	// Populated ID identifies an item in the sorter
	// Between the two Divert status codes indicates that the item has attempted to divert
	IF ExitItemInSorter.ID <> '' THEN
		// Capture the Item encoder index and the Item at the current index
		//  This represents the first item record for this item
		//  It is captured to log the start index to allow this first record to be updated
		//  when the item is completely diverted
		IF ExitItemFound.Item.ID = '' THEN
			ExitItemFound.Counts := ExitSorterIndex;
			ExitItemFound.Item := ExitItemInSorter;
			IF ExitItemFound.Item.Status = E_StatusCode.Divert_Complete THEN
				ExitComplete := TRUE;
			END_IF
		END_IF
		// When ExitComplete is TRUE, and the ID's match, clear out this Item
		IF ExitComplete THEN
			IF ExitItemInSorter.ID = ExitItemFound.Item.ID THEN
				IF aItems[ExitSorterIndex].ID <> '' THEN
					IF .nSortBufferLogEnable.BUFFER_DUMP THEN
						sMessage := CONCAT(' Item: ', aItems[ExitSorterIndex].ID);
						sMessage := CONCAT(sMessage,' Index: ');
						sMessage := CONCAT(sMessage, UDINT_TO_STRING(ExitSorterIndex));
						sMessage := CONCAT(sMessage,' Item Status: ');
						sMessage := CONCAT(sMessage, DINT_TO_STRING(aItems[ExitSorterIndex].Status));
						sMessage := CONCAT(sMessage,' Item Ext Status: ');
						sMessage := CONCAT(sMessage, DINT_TO_STRING(aItems[ExitSorterIndex].ExtStatus));
						// Write to the Error List
						ADSLOGSTR( msgCtrlMask := ADSLOG_MSGTYPE_HINT OR ADSLOG_MSGTYPE_LOG
							, msgFmtStr := 'Exit Complete Dump Info: %s'
							, strArg := sMessage);
					END_IF
				END_IF
				aItems[ExitSorterIndex] := BlankItem;
			END_IF
		// When ExitComplete is FALSE, test for a diverting/diverted item
		ELSE
			// Detect when this item is in a diverting state
			IF (ExitItemInSorter.Status >= E_StatusCode.Diverting
			   OR ExitItemInSorter.Status <= E_StatusCode.Divert_Success)
			   THEN
			   	ExitInDivert := TRUE;
				(*
					Status value increase from Diverting to Divert_Complete
					Codes to indicate divert disposition are between Diverting and Divert_Detected
					Divert_Full and Diverting are set in FB_DivertDecision/FB_DivertControl
					Divert_Detected, Divert_Success, and Divert_Missed are set in FB_ConfirmCheck
				*)
				ExitDiverting := TRUE;
				IF ExitItemInSorter.Status = E_StatusCode.Divert_Detected THEN
					ExitDetected := TRUE;
				END_IF
				// Once the divert is successful, we are no longer "diverting"
				IF ExitItemInSorter.Status = E_StatusCode.Divert_Success THEN
					ExitSuccess := TRUE;
					ExitDiverting := FALSE;
				END_IF
				(*	
					ExitItemInSorter is the current item being examined
					ExitItemFound.Item is a copy of the Array item at ExitItemFound.Counts
					ExitItemFound.Counts references the Array index of the first record associated with this item
					When a Status/ExtStatus of greater value is detected, the first record Status/ExtStatus is overwritten
					The ExitItemFound.Item.Status/.ExtStatus is also updated
				*)
				IF ExitItemInSorter.Status > aItems[ExitItemFound.Counts].Status THEN
					aItems[ExitItemFound.Counts].Status := ExitItemInSorter.Status;
					ExitItemFound.Item.Status := ExitItemInSorter.Status;
				END_IF
				IF ExitItemInSorter.ExtStatus > aItems[ExitItemFound.Counts].ExtStatus THEN
					aItems[ExitItemFound.Counts].ExtStatus := ExitItemInSorter.ExtStatus;
					ExitItemFound.Item.ExtStatus := ExitItemInSorter.ExtStatus;
				END_IF
			END_IF
			aItems[ExitSorterIndex].Status := ExitItemFound.Item.Status;
		END_IF
	ELSE
		(*
			This path is followed when the ExitItemInSorter.ID is empty, which indicates
			that the array record associated with this index is not occupied

			ExitInDivert, ExitDiverting and ExitSuccess are all set while the .ID is not empty
		*)
		// This item was in a "diverting" state
		IF ExitInDivert THEN
			// This item is not currently diverting
			IF NOT ExitDiverting THEN
				// Only change to a Divert_Success if a Divert_Success was detected
				// Any other status is captured in the ELSE clause of the CASE statement
				IF ExitSuccess THEN
					ExitItemFound.Item.Status := E_StatusCode.Divert_Success;
				END_IF
				ExitItemFound.Item.CapturedInMetrics := TRUE;
				ExitItemFound.Item.MessageType := E_MessageIds.TransportComplete_26;
				fb_UpdateBuffer.AddItem(ExitItemFound.Item);
				aItems[ExitItemFound.Counts].Status := E_StatusCode.Divert_Complete;
			END_IF
		END_IF
		// Clear the last detected Exit item
		ExitItemFound.Item := BlankItem;
		// Reset the Detection booleans
		ExitInDivert := FALSE;
		ExitDiverting := FALSE;
		ExitDetected := FALSE;
		ExitSuccess := FALSE;
		ExitComplete := FALSE;
	END_IF
END_FOR

// If the ID is populated, we didn't find a match to update
IF st_ToUpdate.Item.ID <> '' THEN
	IF .nSortBufferLogEnable.BUFFER_UNASSIGNED THEN
		sMessage := CONCAT(' Item: ', st_ToUpdate.Item.ID);
		// Write to the Error List
		ADSLOGSTR( msgCtrlMask := ADSLOG_MSGTYPE_HINT OR ADSLOG_MSGTYPE_LOG
			, msgFmtStr := 'Item Not Updated: %s'
			, strArg := sMessage);
	END_IF
	st_ToUpdate.Item.Status := E_StatusCode.Assign_NotFound;
	st_ToUpdate.Item.DeviceID := st_Sorter.Config.Name;
	st_ToUpdate.Item.MessageType := E_MessageIds.TransportResponse_25;
	fb_UpDateBuffer.AddItem(st_ItemToAdd := st_ToUpdate.Item);
	st_ToUpdate.Item := BlankItem;
END_IF

END_PROGRAM

// ---- POUs/Sorter_P2150.TcPOU
PROGRAM Sorter_P2150

VAR_IN_OUT
	In_ItemToInduct					: ST_Item;
	In_InductingItem				: ST_Item;
	st_tempItem						: ST_ItemTemporary;	// Temporary record used when barcode not yet received
	{attribute 'OPC.UA.DA' := '0'}
	st_Sorter						: ST_Sorter;
	{attribute 'OPC.UA.DA' := '0'}
	aDiverts						: ARRAY[Sorter.DIVERTMIN_P2150..Sorter.NUMBEROFDIVERTS_P2150] OF ST_DIVERT;
	aItems 							: ARRAY[Sorter.SORTERENCODERMIN_P2150..Sorter.SORTERENCODERMAX_P2150] OF ST_Item;
END_VAR

VAR_INPUT
	DestinationOverride	: DINT;	// Pass in Divert to sent item to regardless of the direction received
	ItemsArrayMax		: UDINT;
	ItemsArrayMin		: UDINT;
	DivertArrayMax		: DINT;
	DivertArrayMin		: DINT;
END_VAR

VAR_OUTPUT
	st_DischargeItem	:	ST_Item;
END_VAR
VAR
	// Sorter Diagnostics
	aSorterDiagLog		: ST_ItemLogBuffer;
	fbSorterDiagLog		: FB_ItemLogBuffer;

	//Logging Variables
	UpdateSorterLog : FB_UpdateLog;
	
	//Induct Variables
	testEncoderCount		: UDINT;
	exitEncoderCount		: UDINT;
	lastCompareCount		: UDINT;
	updatingEncoderCount	: UDINT;

	tailendcount		: DINT := 0;
	inductindex 		: DINT;
	
	//Divert Variables
	{attribute 'OPC.UA.DA' := '0'}
	fb_DivertDecision 		: FB_DivertDecision;
	{attribute 'OPC.UA.DA' := '0'}
	fb_DivertFullMonitor  	: ARRAY[Sorter.DIVERTMIN_P2150..Sorter.NUMBEROFDIVERTS_P2150] OF FB_DivertFullMonitor;
	DivertIndex				: DINT;
	Divertoffset			: INT;
	nTestItemIndex			: UDINT;
	Output2ItemIndex		: UDINT;

	// Confirm Check variables
	fb_ConfirmCheck 		: ARRAY[Sorter.DIVERTMIN_P2150..Sorter.NUMBEROFDIVERTS_P2150] OF FB_ConfirmCheck;
	st_ConfirmItem 			: ARRAY[Sorter.DIVERTMIN_P2150..Sorter.NUMBEROFDIVERTS_P2150] OF ST_Item;
	nConfirmItemIndex 		: UDINT;
	
	workingItem			: ST_Item;	// Actual item to induct

	LastItemInducted 	: STRING;
	nIndexToClear		: UDINT;	// Clear Item Array at this index
	nItemArraySize		: UDINT;

	rInductPE			: R_TRIG; 	// Capture the Rising edge of the Induct PE
	fInductPE			: F_TRIG; 	// Capture the Falling edge of the Induct PE
	sMessage			: STRING;

	st_DisplayItem		:st_Item;
	
	LogSorterDump: BOOL := FALSE;

	fb_FindDestination		: FB_FindDestination;
	{attribute 'OPC.UA.DA' := '0'}
	aTempDiverts			: ARRAY[Sorter.DIVERTMIN_P2150..Sorter.NUMBEROFDIVERTS_P2150] OF ST_DIVERT;

	nItemBufferLogEnable	:	UDINT;
	nSorterLogEnable		:	UDINT;
	nDivertLogEnable		:	UDINT;
	nSortBufferLogEnable	:	UDINT;
END_VAR

nItemBufferLogEnable := GVL_Logging.nItemBufferLogEnable OR GVL_Logging.nItemBufferLogEnableP2150;
nSorterLogEnable := GVL_Logging.nSorterLogEnable OR GVL_Logging.nSorterLogEnableP2150;
nDivertLogEnable := GVL_Logging.nDivertLogEnable OR GVL_Logging.nDivertLogEnableP2150;
nSortBufferLogEnable := GVL_Logging.nSortBufferLogEnable OR GVL_Logging.nSortBufferLogEnableP2150;
aTempDiverts := aDiverts;

// Initialize FB_ItemExtBuffer
fbSorterDiagLog(st_BufferData := aSorterDiagLog);

(*
// Test visu variables	
inductPE := SorterInductPE;
ItemsOut := Items;
ArrivalOut := ArrivalBuffer;
// End test variables
*)
(*
	Capture the Upper/Lower bound of relevant IO_OUT arrays for looping purposes
	ItemsArrayMax/Min for the sorter array slot count
*)
// Size is Max - Min + 1 to capture both extremes
nItemArraySize := ItemsArrayMax - ItemsArrayMin + 1;

FOR divertIndex := DivertArrayMin TO DivertArrayMax DO
	fb_DivertFullMonitor[DivertIndex](Divert := aDiverts[divertIndex]);
END_FOR

(*
	Detect barcode receipt after item is already in Item array
	the tempItem is reset when the induct PE is cleared
	The tempItem is populated when the induct PE is blocked and there
	is not an associated barcode waiting to be inducted
*)
IF st_tempItem.Item.ID <> '' THEN
	// Test the IN_ItemToInduct.ID for a value
	// This record will be cleared as soon as it reaches the sorter loop
	IF In_ItemToInduct.ID <> '' THEN
		// The tempItem is overwritten with the IN_ItemToInduct after it is updated
		// But the starting encoder count is not changed so the same items can be updated
		// if the destination update is received while the item is still being inducted
		IF In_ItemToInduct.ID <> st_tempItem.Item.ID THEN 
			// Set the starting count for the testing/updating process
			// The testEncodeCount is incremented upon start, so we start -1 of the encoder count for the item
			testEncoderCount := f_CalculateIndex(Offset := -1, InitialValue:= st_tempItem.Counts, BufferSize := nItemArraySize);
			// Clear the length and start over
			In_ItemToInduct.Length := 0;
			st_tempItem.Item := In_ItemToInduct;
		END_IF 
		// Test for a change of destination after the barcode data has been received
		IF In_ItemToInduct.Destination <> st_tempItem.Item.Destination THEN 
			// Set the starting count for the testing/updating process
			// The testEncodeCount is incremented upon start, so we start -1 of the encoder count for the item
			testEncoderCount := f_CalculateIndex(Offset := -1, InitialValue:= st_tempItem.Counts, BufferSize := nItemArraySize);
			// Clear the length and start over
			In_ItemToInduct.Length := 0;
			// Copy the IN_ItemToInduct to prevent running this until something else in the record changes
			st_tempItem.Item := IN_ItemToInduct;
		END_IF
	END_IF 
END_IF


// Test for the rising edge of the induct PE
// Use this rising edge to log the IN_ItemToInduct record
rInductPE(CLK:= st_Sorter.InductPE, Q =>);

IF rInductPE.Q THEN
	IF nSorterLogEnable.SORTER_INDUCT THEN
		sMessage := CONCAT('Item: ', In_ItemToInduct.ID);
		sMessage := CONCAT(sMessage, ' Pulses: ');
		sMessage := CONCAT(sMessage, UDINT_TO_STRING(st_Sorter.EncoderCounts));
		// Write to the Error List
		ADSLOGSTR( msgCtrlMask := ADSLOG_MSGTYPE_HINT OR ADSLOG_MSGTYPE_LOG
			, msgFmtStr := CONCAT(st_sorter.Config.Name, ' Induct Info: %s')
			, strArg := sMessage);
	END_IF
END_IF
// Test for the falling edge of the induct PE
// Use this falling edge to clear the IN_ItemToInduct record
fInductPE(CLK:= st_Sorter.InductPE, Q =>);

IF fInductPE.Q THEN
	IF nSorterLogEnable.SORTER_INDUCT THEN
		sMessage := CONCAT('Item: ', In_ItemToInduct.ID);
		sMessage := CONCAT(sMessage,' Pulses: ');
		sMessage := CONCAT(sMEssage, UDINT_TO_STRING(st_Sorter.EncoderCounts));
		// Write to the Error List
		ADSLOGSTR( msgCtrlMask := ADSLOG_MSGTYPE_HINT OR ADSLOG_MSGTYPE_LOG
			, msgFmtStr := CONCAT(st_sorter.Config.Name, ' Cleared Induct Info: %s')
			, strArg := sMessage);
	END_IF
	// Clear the record
	In_InductingItem :=  BlankItem;
END_IF

// Process every array index between the current index and the last processed index
WHILE st_Sorter.EncoderCounts <> testEncoderCount DO

	// Capture the lastEncoderCount before changing it for comparison of last inducted items
	lastCompareCount := testEncoderCount;

	// Increment the testEncoderCount
	// The testEncoderCount variable will be used throughout the processing to ensure
	//	that all array elements are processed
	testEncoderCount := f_CalculateIndex(Offset := 1, InitialValue:= testEncoderCount, BufferSize := nItemArraySize);
	IF st_Sorter.InductPE THEN
	  	IF (In_ItemToInduct.ID <> '') THEN
			In_InductingItem := In_ItemToInduct;
			In_ItemToInduct := BlankItem;
			// If there is an override, use the value as the destination
			IF DestinationOverride <> 0 THEN
				IF nSorterLogEnable.SORTER_DESTINATION_LU THEN
					sMessage := CONCAT(' Orig: ', DINT_TO_STRING(In_InductingItem.Destination));
					sMessage := CONCAT(sMessage, 'New: ');
					sMessage := CONCAT(sMessage, DINT_TO_STRING(DestinationOverride));
					// Write to the Error List
					ADSLOGSTR( msgCtrlMask := ADSLOG_MSGTYPE_HINT OR ADSLOG_MSGTYPE_LOG
						, msgFmtStr := CONCAT(st_sorter.Config.Name, ' DestinationOverride %s')
						, strArg := sMessage);
				END_IF
				In_InductingItem.Destination := DestinationOverride;
			END_IF
			IF nSorterLogEnable.SORTER_DESTINATION_LU THEN
				sMessage := CONCAT('Destination: ', DINT_TO_STRING(In_InductingItem.Destination));
				// Write to the Error List
				ADSLOGSTR( msgCtrlMask := ADSLOG_MSGTYPE_HINT OR ADSLOG_MSGTYPE_LOG
					, msgFmtStr := CONCAT(st_sorter.Config.Name, ' Sorter Lookup %s')
					, strArg := sMessage);
			END_IF
			fb_FindDestination(RoundRobin := st_Sorter.RoundRobin
							, SorterLogEnable := nSorterLogEnable
							, aDiverts := aTempDiverts
							, DestinationID := In_InductingItem.Destination
							, DestinationIndex => In_InductingItem.DestinationIdx);
			IF nSorterLogEnable.SORTER_INDUCT_PE THEN
				sMessage := CONCAT('Item: ', In_InductingItem.ID);
				sMessage := CONCAT(sMessage,' Pulses: ');
				sMessage := CONCAT(sMessage, UDINT_TO_STRING(st_Sorter.EncoderCounts));
				sMessage := CONCAT(sMessage,' Dest: ');
				sMessage := CONCAT(sMessage, DINT_TO_STRING(In_InductingItem.Destination));
				sMessage := CONCAT(sMessage,' DestIdx: ');
				sMessage := CONCAT(sMessage, DINT_TO_STRING(In_InductingItem.DestinationIdx));
				// Write to the Error List
				ADSLOGSTR( msgCtrlMask := ADSLOG_MSGTYPE_HINT OR ADSLOG_MSGTYPE_LOG
					, msgFmtStr := CONCAT(st_sorter.Config.Name, ' Inducting Info: %s')
					, strArg := sMessage);
			END_IF
		END_IF
	  	IF (In_InductingItem.ID <> '') THEN
			LastItemInducted := In_InductingItem.ID;
			IF aItems[testEncoderCount].ID <> '' THEN
				IF aItems[testEncoderCount].Status >= E_StatusCode.Diverting AND aItems[testEncoderCount].Status <= E_StatusCode.Divert_UnknownError THEN
					aItems[testEncoderCount].Status := E_StatusCode.Divert_UnknownError;
				END_IF
				UpdateSorterLog(Status := aItems[testEncoderCount].Status, ItemID := aItems[testEncoderCount].UniqueID);
			END_IF
		
			// Set the Item status
			In_InductingItem.Status := E_StatusCode.In_Sorter;

			// Check for destination full on the first pass, then ignore it.
			IF In_InductingItem.Length = 0 AND DestinationOverride = 0 THEN
				IF aDiverts[In_InductingItem.DestinationIdx].Full AND DestinationOverride = 0 THEN
					IF st_Sorter.Config.RecircUsed THEN
						In_InductingItem.Destination := st_Sorter.Config.RecircDestination;
						In_InductingItem.DestinationIdx := st_Sorter.Config.RecircDestIdx;
						In_InductingItem.ExtStatus := E_StatusCode.Divert_Recirculated;
					ELSE
						In_InductingItem.Destination := st_Sorter.Config.DefaultDestination;
						In_InductingItem.DestinationIdx := st_Sorter.Config.DefaultDestIdx;
						In_InductingItem.ExtStatus := E_StatusCode.Divert_Full;
					END_IF
				END_IF
			END_IF
			// Clear the extend counter
			tailendcount := 0;

			// Copy the ItemToInduct to the WorkingItem that will be inducted
			workingItem := In_InductingItem;
			// Increment the Length on the ItemToInduct record, then it will be added to the array
			//  and the length will increment
			In_InductingItem.Length := In_InductingItem.Length +  1;
			// Determined by UniqueID = 0
		ELSE //If the item makes it to the sorter, but is not identified, induct the item with tempItem.Item
			LastItemInducted := 'UNKNOWN';
			UpdateSorterLog(Status := E_StatusCode.UnidentifiedItem, ItemID := st_tempItem.Item.UniqueID);

			// Process this the first time
			IF st_tempItem.Item.Length = 0 THEN
				IF nSorterLogEnable.SORTER_INDUCT_PE THEN
					sMessage := CONCAT('Temp Item: ', st_tempItem.Item.ID);
					sMessage := CONCAT(sMessage,' Pulses: ');
					sMessage := CONCAT(sMessage, UDINT_TO_STRING(st_Sorter.EncoderCounts));
					sMessage := CONCAT(sMessage,' Dest: ');
					sMessage := CONCAT(sMessage, DINT_TO_STRING(st_tempItem.Item.Destination));
					sMessage := CONCAT(sMessage,' DestIdx: ');
					sMessage := CONCAT(sMessage, DINT_TO_STRING(st_tempItem.Item.DestinationIdx));
					sMessage := CONCAT(sMessage,' Length: ');
					sMessage := CONCAT(sMessage, DINT_TO_STRING(st_tempItem.Item.Length));
					// Write to the Error List
					ADSLOGSTR( msgCtrlMask := ADSLOG_MSGTYPE_HINT OR ADSLOG_MSGTYPE_LOG
						, msgFmtStr := CONCAT(st_sorter.Config.Name, ' Inducting Info: %s')
						, strArg := sMessage);
				END_IF
				IF aDiverts[st_Sorter.Config.DefaultDestIdx].Full THEN
					IF st_Sorter.Config.RecircUsed THEN
						st_tempItem.Item.Destination := st_Sorter.Config.RecircDestination;
						st_tempItem.Item.DestinationIdx := st_Sorter.Config.RecircDestIdx;
						st_tempItem.Item.ExtStatus := E_StatusCode.Divert_Recirculated;
					ELSE
						st_tempItem.Item.Destination := st_Sorter.Config.DefaultDestination;
						st_tempItem.Item.DestinationIdx := st_Sorter.Config.DefaultDestIdx;
						st_tempItem.Item.ExtStatus := E_StatusCode.Divert_Full;
					END_IF
				ELSE
					IF DestinationOverride = 0 THEN
						st_tempItem.Item.Destination := st_Sorter.Config.DefaultDestination;
					ELSE
						st_tempItem.Item.Destination := DestinationOverride;
					END_IF
					IF nSorterLogEnable.SORTER_DESTINATION_LU THEN
						sMessage := CONCAT('Destination: ', DINT_TO_STRING(st_tempItem.Item.Destination));
						// Write to the Error List
						ADSLOGSTR( msgCtrlMask := ADSLOG_MSGTYPE_HINT OR ADSLOG_MSGTYPE_LOG
							, msgFmtStr := CONCAT(st_sorter.Config.Name, ' Temp Lookup %s')
							, strArg := sMessage);
					END_IF
					fb_FindDestination(RoundRobin := st_Sorter.RoundRobin
							, SorterLogEnable := nSorterLogEnable
							, aDiverts := aTempDiverts
							, DestinationID := st_tempItem.Item.Destination
							, DestinationIndex => st_tempItem.Item.DestinationIdx);
				END_IF		
				IF nSorterLogEnable.SORTER_INDUCT_PE THEN
					sMessage := CONCAT('Temp Item: ', st_tempItem.Item.ID);
					sMessage := CONCAT(sMessage,' Pulses: ');
					sMessage := CONCAT(sMessage, UDINT_TO_STRING(st_Sorter.EncoderCounts));
					sMessage := CONCAT(sMessage,' Dest: ');
					sMessage := CONCAT(sMessage, DINT_TO_STRING(st_tempItem.Item.Destination));
					sMessage := CONCAT(sMessage,' DestIdx: ');
					sMessage := CONCAT(sMessage, DINT_TO_STRING(st_tempItem.Item.DestinationIdx));
					// Write to the Error List
					ADSLOGSTR( msgCtrlMask := ADSLOG_MSGTYPE_HINT OR ADSLOG_MSGTYPE_LOG
						, msgFmtStr := CONCAT(st_sorter.Config.Name, ' Inducting Info: %s')
						, strArg := sMessage);
				END_IF
			END_IF
			// Copy the tempItem.Item to the WorkingItem that will be inducted
			workingItem := st_tempItem.Item;
			// Increment the Length on the ItemToInduct record, then it will be added to the array
			//  and the length will increment
			st_tempItem.Item.Length := st_tempItem.Item.Length +  1;
		END_IF

		// Induct everything
		aItems[testEncoderCount] := workingItem;
		fbSorterDiagLog.AddItem(workingItem);
	// Follow this path when the induct photo-eye is cleared
	ELSE
		// Extend the end of the item by a set amount, or to a mimimum length
		// Test to verify that the Item index is clear, and we are still extending the length of the item
		IF aItems[lastCompareCount].ID <> '' THEN
			IF tailendcount < st_Sorter.Config.TailEndLength AND st_Sorter.Config.TailEndLength > 0 THEN
				aItems[testEncoderCount] := aItems[lastCompareCount]; 
				fbSorterDiagLog.AddItem(aItems[lastCompareCount]);
				aItems[testEncoderCount].Length := aItems[testEncoderCount].Length + 1;
				tailendcount := tailendcount + 1;
			END_IF
			IF aItems[lastCompareCount].Length < st_Sorter.Config.MinimumLength AND st_Sorter.Config.MinimumLength > 0 THEN
				aItems[testEncoderCount] := aItems[lastCompareCount]; 
				fbSorterDiagLog.AddItem(aItems[lastCompareCount]);
				aItems[testEncoderCount].Length := aItems[testEncoderCount].Length + 1;
			END_IF
		END_IF
	END_IF
END_WHILE

// Process every array index between the current index and the last processed exit index
WHILE st_Sorter.EncoderCounts <> exitEncoderCount DO

	// Increment the exitEncoderCount
	// The exitEncoderCount variable will be used throughout the processing to ensure
	//	that all array elements are processed
	exitEncoderCount := f_CalculateIndex(Offset := 1, InitialValue:= exitEncoderCount, BufferSize := nItemArraySize);
	// Process the diverts relative to the current encoder count
	FOR divertIndex := DivertArrayMin TO DivertArrayMax DO
		// Get the distance to each divert, distance is the number of pulses to actuation
		Divertoffset := aDiverts[divertIndex].Config.Distance;
		// Calculate the index of the item to test for a divert
		// Subtract the offset from the current encoder count (exitEncoderCount)
		// As the encoder count increases, the current index pointer advances
		// Subtracting looks backwards into the sorter item array to test for items at the diverts
		//	distance that should be diverted
		nTestItemIndex := F_CalculateIndex(initialvalue := exitEncoderCount
										, offset := -(Divertoffset)
										, BufferSize := (ItemsArrayMax + 1));	
		//Setup Out2Item for energizing 2nd divert output
		Output2ItemIndex := F_CalculateIndex(initialvalue := exitEncoderCount
										, offset := -(Divertoffset + UINT_TO_INT(st_Sorter.Config.Output2Offset))
										, BufferSize := (ItemsArrayMax + 1));	
		// Log Diverts
		IF aItems[nTestItemIndex].DestinationIdx = divertIndex THEN
			IF nSorterLogEnable.SORTER_DIVERTS THEN
				sMessage := CONCAT('Item: ', aItems[nTestItemIndex].ID);
				sMessage := CONCAT(sMessage,' Index: ');
				sMessage := CONCAT(sMessage, UDINT_TO_STRING(nTestItemIndex));
				sMessage := CONCAT(sMessage,' Dest: ');
				sMessage := CONCAT(sMessage, DINT_TO_STRING(aItems[nTestItemIndex].Destination));
				sMessage := CONCAT(sMessage,' DestIdx: ');
				sMessage := CONCAT(sMessage, DINT_TO_STRING(aItems[nTestItemIndex].DestinationIdx));
				sMessage := CONCAT(sMessage,' Divert Status: ');
				sMessage := CONCAT(sMessage, DINT_TO_STRING(aDiverts[DivertIndex].Status));
				sMessage := CONCAT(sMessage,' Item Status: ');
				sMessage := CONCAT(sMessage, DINT_TO_STRING(aItems[nTestItemIndex].Status));
				// Write to the Error List
				ADSLOGSTR( msgCtrlMask := ADSLOG_MSGTYPE_HINT OR ADSLOG_MSGTYPE_LOG
					, msgFmtStr := CONCAT(st_sorter.Config.Name, ' Item at Divert Index: %s')
					, strArg := sMessage);
			END_IF
		END_IF
		fb_DivertDecision( bLog := nDivertLogEnable.DIVERT_DECISION 
					 , Output1Item		:= aItems[nTestItemIndex]
					 , Output2Item		:= aItems[Output2ItemIndex]
					 , Divert 			:= aDiverts[DivertIndex]
					 , DivertIndex		:= DivertIndex
					 );
		// Calculate the distance to the confirm PE to test for a successful divert
		nConfirmItemIndex := F_CalculateIndex(initialvalue := exitEncoderCount
										, offset := -(Divertoffset + aDiverts[divertIndex].Config.ConfirmDist)
										, BufferSize := (ItemsArrayMax + 1));
		// Log Confirms
		IF aItems[nConfirmItemIndex].Status >= E_StatusCode.Diverting
		   AND aItems[nConfirmItemIndex].Status <= E_StatusCode.Divert_Complete
		   AND aItems[nConfirmItemIndex].UniqueID <> 0
		   AND aItems[nConfirmItemIndex].DestinationIdx = DivertIndex
		   THEN
			IF nSorterLogEnable.SORTER_CONFIRMS THEN
				sMessage := CONCAT('Item: ', aItems[nConfirmItemIndex].ID);
				sMessage := CONCAT(sMessage,' Index: ');
				sMessage := CONCAT(sMessage, UDINT_TO_STRING(nConfirmItemIndex));
				sMessage := CONCAT(sMessage,' Dest: ');
				sMessage := CONCAT(sMessage, DINT_TO_STRING(aItems[nConfirmItemIndex].Destination));
				sMessage := CONCAT(sMessage,' DestIdx: ');
				sMessage := CONCAT(sMessage, DINT_TO_STRING(aItems[nConfirmItemIndex].DestinationIdx));
				sMessage := CONCAT(sMessage,' Divert Status: ');
				sMessage := CONCAT(sMessage, DINT_TO_STRING(aDiverts[DivertIndex].Status));
				sMessage := CONCAT(sMessage,' Item Status: ');
				sMessage := CONCAT(sMessage, DINT_TO_STRING(aItems[nTestItemIndex].Status));
				// Write to the Error List
				ADSLOGSTR( msgCtrlMask := ADSLOG_MSGTYPE_HINT OR ADSLOG_MSGTYPE_LOG
					, msgFmtStr := CONCAT(st_sorter.Config.Name, ' Item at Confirm Index: %s')
					, strArg := sMessage);
			END_IF
		END_IF
		fb_ConfirmCheck[divertIndex] ( bLog := nDivertLogEnable.DIVERT_DECISION 
					 , ConfirmItem		:= aItems[nConfirmItemIndex]
					 , ConfirmPE 		:= aDiverts[DivertIndex].ConfirmPE
					 , DivertIndex		:= DivertIndex
					 , bIsDischarge		:= aDiverts[DivertIndex].Config.IsDischarge
					 , DetectedItem => st_ConfirmItem[DivertIndex]
					 );
	END_FOR
	
	// Capture the last item discharged by this sorter section
	IF st_ConfirmItem[DivertArrayMax].ID <> '' THEN
		st_DischargeItem := st_ConfirmItem[DivertArrayMax];
	END_IF

	// Clear the Item array ahead of the current encoder count
	nIndexToClear := f_CalculateIndex(Offset := 40, InitialValue:= exitEncoderCount, BufferSize := nItemArraySize);
	IF aItems[nIndexToClear].ID <> '' THEN
		IF nSorterLogEnable.SORTER_DUMP THEN
			sMessage := CONCAT('Item: ', aItems[nIndexToClear].ID);
			sMessage := CONCAT(sMessage,' Index: ');
			sMessage := CONCAT(sMessage, UDINT_TO_STRING(nIndexToClear));
			sMessage := CONCAT(sMessage,' Item Status: ');
			sMessage := CONCAT(sMessage, DINT_TO_STRING(aItems[nIndexToClear].Status));
			sMessage := CONCAT(sMessage,' Destination: ');
			sMessage := CONCAT(sMessage, DINT_TO_STRING(aItems[nIndexToClear].Destination));
			sMessage := CONCAT(sMessage,' DestIndex: ');
			sMessage := CONCAT(sMessage, DINT_TO_STRING(aItems[nIndexToClear].DestinationIDX));
			// Write to the Error List
			ADSLOGSTR( msgCtrlMask := ADSLOG_MSGTYPE_HINT OR ADSLOG_MSGTYPE_LOG
				, msgFmtStr := CONCAT(st_sorter.Config.Name, ' Clear Ahead Dump Info: %s')
				, strArg := sMessage);
		END_IF
	END_IF
	aItems[nIndexToClear] := BlankItem;

END_WHILE

END_PROGRAM

// ---- POUs/MsgControl.TcPOU
PROGRAM MsgControl
VAR_INPUT
	TransmitEnable 				: BOOL;
	nConnectionIndex			: UDINT	:= 1;
END_VAR
VAR
	MsgID						: DINT;			// TCP/IP Message ID as per Communication protocol defined in FA 
	DeviceID					: STRING(5);	// TCP/IP Device ID as per Communication protocol defined in FA 
	BarCode						: STRING(20);	// TCP/IP Load ID (Bar Code) as per Communication protocol defined in FA
	BarCodeNoSpace				: STRING(20);	// TCP/IP Load ID (Bar Code) as per Communication protocol defined in FA stripped of spaces  
	Destination					: DINT;			// TCP/IP Destination as per Communication protocol defined in FA
	DefDestination				: DINT;			// TCP/IP Default Destination as per Communication protocol defined in FA
	Status						: BYTE;				// 
	Msg_EquipStatArry			: ARRAY[1..7] OF ST_Msg_EquipStat;
	nSystemStatusIndex 			: DINT; 	// Index used for Processing the system status array
	nTempOperState 				: DINT;	//Capture the Temporary Operating State of the Equipment for comparison
	nEquipStatusIndex			: DINT;	//Index used for adding items to the MSG_EquipStatArray
	StrStartPos					: INT;
	StrEndPos					: INT;
	MsgString					: STRING(55);
	RawMsgArray					: ARRAY[1..10] OF T_MaxString;	// Capture the last Raw messages for troubleshooting
	RawMsgLenArray				: ARRAY[1..10] OF INT;			// Capture the last  Raw message lengths for troubleshooting
	RawMsgStartPosArray			: ARRAY[1..10] OF INT;			// Capture the last  Raw message start positions for troubleshooting
	RawMsgEndPosArray			: ARRAY[1..10] OF INT;			// Capture the last  Raw message end positions for troubleshooting
	MsgArray					: ARRAY[1..10] OF STRING(55);		// Capture the last 10 messages that have been stripped from the starting character  for troubleshooting
	Blank_Msg_ConveyorStatArry	: ARRAY [1..7] OF ST_Msg_EquipStat := [7((Status := 99))];

	i 							: INT;
	j							: INT;
	
	RxCounter_Old				: UDINT;
	TxCounter_Old				: UDINT;
	TransmitMsgBuffer			: ARRAY [1..TransmitMsgBuffer_Size] OF STRING(55);	// Buffer to hold transmit messages
	TransmitMsgBuffer_Index		: INT :=	1;		// Index to the Buffer
	TransmitMsgStatus			: INT;			
	SendingMsg_Index			: INT :=	1;		// Index to send message
	
	ItemTransport				: ST_Item;		// Output Item Update with destination from ARUP Host (Send to Sorter PLC)
	BlankItem					: ST_Item := (ID := '', UniqueID := 0
													, Destination := 0
													, Status := E_StatusCode.No_Status
													, ExtStatus := E_StatusCode.No_Status
													, DeviceID := ''
													, MessageType := E_MessageIds.NoMessage_00);

	ReadBCRID_S2140_01_Old			: UDINT;		// Bar Code watch variable
	ReadBCRID_S2141_01_Old			: UDINT;		// Bar Code watch variable
	ReadBCRID_S2150_01_Old			: UDINT;		// Bar Code watch variable	
	ReadBCRID_S3080_01_Old			: UDINT;		// Bar Code watch variable
			
	TransmittedArray			: ARRAY[0..10] OF STRING(55);
	x							: DINT;
	y							: INT;
	
	SpacePosition				: INT;
	
	fb_CheckStopRegister		: FB_ManageCodes;	// Used to test for a specific Stop Code to report to the Host
	bOverHeight					: BOOL; 	// Detect OverHeight to report to the Host
	st_UpdateMessageToSend		: ST_Item;			// Message to Send to Host

	fb_SorterUpdateBuffer			: FB_ItemBuffer;	// Function to Process the SorterUpdateBuffer

	fb_SorterTransportBuffer_P2140	: FB_ItemBuffer;	// Function to Process the SorterTransportBuffer
	fb_SorterTransportBuffer_P2150	: FB_ItemBuffer;	// Function to Process the SorterTransportBuffer

	sMessage	:	STRING;
	
END_VAR

VAR CONSTANT
	SEND_ARRIVAL			:	INT := 5;
	SEND_LOCATION			:	INT := 7;
	TransmitMsgBuffer_Size	:	INT :=	25;		// Number of Messages to hold in buffer
END_VAR

// Create instances of Buffer Processing Functions to initialize the buffers and data
fb_SorterUpdateBuffer.Master := TRUE;
fb_SorterTransportBuffer_P2140.Master := TRUE;
fb_SorterTransportBuffer_P2150.Master := TRUE;

// Activate or de-activate logging
fb_SorterUpdateBuffer.LogEntries := .nItemBufferLogEnable.UPDATE OR .nItemBufferLogEnableP2150.UPDATE OR .nItemBufferLogEnableP2150.UPDATE;
fb_SorterTransportBuffer_P2140.LogEntries := .nItemBufferLogEnable.TRANSPORT OR .nItemBufferLogEnableP2140.TRANSPORT;
fb_SorterTransportBuffer_P2150.LogEntries := .nItemBufferLogEnable.TRANSPORT OR .nItemBufferLogEnableP2150.TRANSPORT;

// Setup Buffer names for Logging purposes
fb_SorterUpdateBuffer.Name := 'SYS UPDATE';
fb_SorterTransportBuffer_P2140.Name := 'P2140 SYS TRANSPORT';
fb_SorterTransportBuffer_P2150.Name := 'P2150 SYS TRANSPORT';

fb_SorterUpdateBuffer(st_BufferData := st_SorterUpdateBuffer
					, st_BufferFdbkIn := st_UpdateFdbkIn
					, st_BufferFdbkOut => st_UpdateFdbkOut);
fb_SorterTransportBuffer_P2140(st_BufferData := st_SorterTransportBuffer_P2140
					, st_BufferFdbkIn := st_TransportFdbkIn_P2140
					, st_BufferFdbkOut => st_TransportFdbkOut_P2140);
fb_SorterTransportBuffer_P2150(st_BufferData := st_SorterTransportBuffer_P2150
					, st_BufferFdbkIn := st_TransportFdbkIn_P2150
					, st_BufferFdbkOut => st_TransportFdbkOut_P2150);

(* -------------------- On Receive Message Process the data -------------------- *)
IF RxCounter_Old <> ServerControl.fbServer.aApplications[nConnectionIndex].RxCounter  THEN
	ItemTransport := BlankItem; // Clear the ItemTransport each pass to capture only new transport commands
	RECEIVE();
	// Test the DeviceID and route the Transport accordingly
	//	If there is only one possible DeviceID, this IF statement can be removed, but the fb_(TransportBuffer).AddItem call still has to be made
	//	Also, the default destination needs to be passed per DeviceID
	IF DeviceID = Sorter.st_Sorter_P2140Cfg.EquipID THEN
		fb_SorterTransportBuffer_P2140.AddItem(st_ItemToAdd := ItemTransport);
		P2140_DefaultDestination := DefDestination;
	END_IF
	IF DeviceID = Sorter.st_Sorter_P2150Cfg.EquipID THEN
		fb_SorterTransportBuffer_P2150.AddItem(st_ItemToAdd := ItemTransport);
		P2150_DefaultDestination := DefDestination;
	END_IF

	RxCounter_Old := ServerControl.fbServer.aApplications[nConnectionIndex].RxCounter;
END_IF

(* -------------------- Transmit Messages if any are waiting in the buffer --------------------- *)
IF SendingMsg_Index <> TransmitMsgBuffer_Index THEN
	TRANSMIT(TransmitEnable:= TRUE);
END_IF

(* -------------------- Watch Bar code readers and send message when load is read -------------------- *)
(* ----- BCR_S2140_01: P2140 Divert  ----- *)	
ReadBCRID_S2140_01_Old := BarCodeMessage(cDatamanReader := BarCodeReaders.BCR_S2140_01
									, nOldCount := ReadBCRID_S2140_01_Old
									, nMessageToSend := SEND_ARRIVAL);
(* ----- BCR_S2141_01: P2143 Induct Confirm ----- *)	
ReadBCRID_S2141_01_Old := BarCodeMessage(cDatamanReader := BarCodeReaders.BCR_S2141_01
									, nOldCount := ReadBCRID_S2141_01_Old
									, nMessageToSend := SEND_LOCATION);
(* ----- BCR_S2150_01: P2150 Sorter ----- *)	
ReadBCRID_S2150_01_Old := BarCodeMessage(cDatamanReader := BarCodeReaders.BCR_S2150_01
									, nOldCount := ReadBCRID_S2150_01_Old
									, nMessageToSend := SEND_ARRIVAL);
(* ----- BCR_S3080_01: P3080 Lane Confirm ----- *)	
ReadBCRID_S3080_01_Old := BarCodeMessage(cDatamanReader := BarCodeReaders.BCR_S3080_01
									, nOldCount := ReadBCRID_S3080_01_Old
									, nMessageToSend := SEND_LOCATION);


(* -------------------- Watch Sorter and Device Status and transmit on change -------------------- *)
// Transmit On update from Sorter
// Detect a new message to process when the in and out pointer values disagree
IF st_SorterUpdateBuffer.nInPointer <> fb_SorterUpdateBuffer.OutPointer THEN
	// Pull the next message out of the buffer
	fb_SorterUpdateBuffer.RemoveItem(st_ItemToReturn => st_UpdateMessageToSend);
	CASE st_UpdateMessageToSend.MessageType OF

		E_MessageIds.TransportResponse_25:			// Response to a Transport Command

			CASE st_UpdateMessageToSend.Status OF
				E_StatusCode.Assign_Accepted:		// Assignment Accepted
					TransmitMsgStatus := E_TransportResponse.Accepted; 
				E_StatusCode.Assign_Full:			// Assigned Lane Unavailable
					TransmitMsgStatus := E_TransportResponse.DivertLaneUnavailable; 
				E_StatusCode.Assign_NotFound:		// Assigned Load ID Not Found
					TransmitMsgStatus := E_TransportResponse.LoadIdNotFound; 
				E_StatusCode.Assign_NotInducted:	// Assigned Load Not Inducted
					TransmitMsgStatus := E_TransportResponse.NextLoadReady; 
				E_StatusCode.Diverting:	// Assigned Load already Inducting
					TransmitMsgStatus := E_TransportResponse.LateInduction; 
			ELSE
				TransmitMsgStatus := E_TransportResponse.UnknownFailure; // Capture any other failures
				IF nMessageLogEnable.TransportResponse_25 THEN
					sMessage := CONCAT(' Item: ', st_UpdateMessageToSend.ID);
					sMessage := CONCAT(sMessage,' Destination: ');
					sMessage := CONCAT(sMessage, DINT_TO_STRING(st_UpdateMessageToSend.Destination));
					sMessage := CONCAT(sMessage,' TR Status: ');
					sMessage := CONCAT(sMessage, DINT_TO_STRING(st_UpdateMessageToSend.Status));
					// Write to the Error List
					ADSLOGSTR( msgCtrlMask := ADSLOG_MSGTYPE_HINT OR ADSLOG_MSGTYPE_LOG
						, msgFmtStr := 'Unhandled Transport Response Status: %s'
						, strArg := sMessage);
				END_IF
			END_CASE
			TransmitMsgBuffer[TransmitMsgBuffer_Index] := TransportResponse(Device := st_UpdateMessageToSend.DeviceID
																			, Barcode := st_UpdateMessageToSend.ID
																			, Status := TransmitMsgStatus);
			TransmitMsgBuffer_Index := IncIndex(TransmitMsgBuffer_Index,1,TransmitMsgBuffer_Size);

		E_MessageIds.TransportComplete_26:			// Indication of the final disposition of a transported item

			CASE st_UpdateMessageToSend.Status OF
				E_StatusCode.Divert_Success:		// Divert Success Message
					TransmitMsgStatus := E_TransportComplete.Success; 
				E_StatusCode.Divert_Complete:		// Divert Success Message
					TransmitMsgStatus := E_TransportComplete.Success; 
			ELSE 									// Catch all other failures
				TransmitMsgStatus := E_TransportComplete.Faulted; 
			END_CASE			
			CASE st_UpdateMessageToSend.ExtStatus OF
				E_StatusCode.Divert_Full:			// Divert Full/Unavailable
					TransmitMsgStatus := E_TransportComplete.Unavailable; 
				E_StatusCode.Divert_Offline:		// Divert Offline
					TransmitMsgStatus := E_TransportComplete.Offline; 
				E_StatusCode.Divert_Missed:		// Divert Missed
					TransmitMsgStatus := E_TransportComplete.Passed; 
				E_StatusCode.Divert_Recirculated:		// Divert Missed
					TransmitMsgStatus := E_TransportComplete.Success; 
			END_CASE			
			TransmitMsgBuffer[TransmitMsgBuffer_Index] := TransportComplete(Device:= st_UpdateMessageToSend.DeviceID
																			, BarCode:= st_UpdateMessageToSend.ID
																			, Dest:= DINT_TO_INT(st_UpdateMessageToSend.Destination)
																			, Status:= TransmitMsgStatus ); 
			TransmitMsgBuffer_Index := IncIndex(TransmitMsgBuffer_Index,1,TransmitMsgBuffer_Size);

	END_CASE
END_IF

// Transmit on Device Status Change
DeviceStatus();

(* -------------------- Reset The Transmit Triger after the message is succesfully added to the buffer ------------------- *)
IF ((ServerControl.fbServer.aApplications[nConnectionIndex].bTransmitTrigger = TRUE) OR ServerControl.TransmitTrigger = TRUE)  AND (TxCounter_Old <> ServerControl.fbServer.aApplications[nConnectionIndex].TxCounter) THEN
	ServerControl.TransmitTrigger := FALSE;
	TRANSMIT(TransmitEnable:= FALSE);
	TxCounter_Old := ServerControl.fbServer.aApplications[nConnectionIndex].TxCounter;
END_IF

METHOD PRIVATE Arrival : STRING(55)
VAR_INPUT
	Device :	STRING(5);		// Device Label per communication standard
	BarCode:	STRING(30);		// Barcode from barcode reader
	DefDest:	INT;		// Default destination
END_VAR
VAR
	String1: STRING(55);
	BC_Len: INT;
	x: INT;
	String_DefDest: STRING(2);
	y: INT;
	Device_Len: INT;
	i: INT;
END_VAR
(* Message from communication Spec:
	[STX (0x02h)][23][Device ID (5 CHR)][Barcode (20 CHR)][Default Dest (2 CHR)][Blank (22 CHR)][ETX 0x03h)]
*)

// Start Message with header
String1 := '$0223';

// Check Device for length and Pad with spaces if needed
Device_Len := LEN(Device);
IF Device_Len = 5 THEN
	String1 := CONCAT(STRING1, Device);
ELSIF Device_Len < 5 THEN
	String1 := CONCAT(STRING1, Device);
	FOR i := 1 TO (5-Device_Len) DO
		String1 := CONCAT(String1,' ');
	END_FOR
ELSE
	String1 := CONCAT(String1, 'XXXXX');
END_IF

// Check Barcode for length and Pad with spaces if needed
BC_Len := LEN(BARCODE);
IF BC_Len <20 THEN
	String1 := CONCAT(STRING1, BarCode);
	FOR x := 1 TO (20-BC_Len) DO
		String1 := CONCAT(String1,' ');
	END_FOR
ELSIF BC_Len = 20 THEN
	String1 := CONCAT(STRING1, BarCode);
ELSE 
	String1 := CONCAT(STRING1, RIGHT(BarCode,20));	
END_IF

// Check Default Destination for length and Pad with spaces if needed
String_DefDest := INT_TO_STRING(DefDest);
IF DefDest < 10 THEN
	String1 := CONCAT(String1,'0');
	String1 := CONCAT(String1, String_DefDest);
ELSIF (DefDest >= 10) AND (DefDest < 100) THEN
	String1 := CONCAT(String1, String_DefDest);
ELSE
	String1 := CONCAT(String1, 'XX');
END_IF	

// Pad with spaces
FOR y := 1 TO 22 DO
	String1 := CONCAT(String1,' ');
END_FOR

// Add ending Character
String1 := CONCAT(String1,'$03');
	
Arrival := String1;
END_METHOD

METHOD PRIVATE BarCodeMessage : UDINT
VAR_INPUT
	cDatamanReader	: CognexDataMan260;
//	sLocation		:	STRING(5);
	nOldCount		:	UDINT;
	nMessageToSend	: 	INT;
END_VAR
IF nOldCount <> cDatamanReader.GoodreadCount THEN
	// Send location update message to host
	CASE nMessageToSend OF
		SEND_ARRIVAL:	TransmitMsgBuffer[TransmitMsgBuffer_Index] := Arrival(cDatamanReader.In_EquipID, cDatamanReader.Out_ReadString,00);
		SEND_LOCATION: TransmitMsgBuffer[TransmitMsgBuffer_Index] := LocationUpdate(cDatamanReader.In_EquipID, cDatamanReader.Out_ReadString,00);
	END_CASE
	TransmitMsgBuffer_Index := IncIndex(TransmitMsgBuffer_Index,1,TransmitMsgBuffer_Size);
	BarCodeMessage := cDatamanReader.GoodreadCount;
ELSE
	BarCodeMessage := nOldCount;
END_IF
END_METHOD

METHOD PRIVATE CustomMessage : UDINT
VAR_INPUT
	EquipID			: 	STRING(5);
	Barcode			:	STRING(30);
	nReadCount		:	UDINT;
	nOldCount		:	UDINT;
	nMessageToSend	: 	INT;
END_VAR
IF nOldCount <> nReadCount THEN
	// Send location update message to host
	CASE nMessageToSend OF
		SEND_ARRIVAL:	TransmitMsgBuffer[TransmitMsgBuffer_Index] := Arrival(EquipID, BarCode,00);
		SEND_LOCATION: TransmitMsgBuffer[TransmitMsgBuffer_Index] := LocationUpdate(EquipID, BarCode,00);
	END_CASE
	TransmitMsgBuffer_Index := IncIndex(TransmitMsgBuffer_Index,1,TransmitMsgBuffer_Size);
	CustomMessage := nReadCount;
ELSE
	CustomMessage := nOldCount;
END_IF
END_METHOD

ACTION DeviceStatus:
(*
	
	Local Data items used for Equipment status processing
	Msg_EquipStatArry:	ARRAY[1..7] OF ST_Msg_EquipStat;
	nSystemStatusIndex : INT; 	// Index used for Processing the system status array
	nEquipStatusIndex: INT;	//Index used for adding items to the MSG_EquipStatArray
	nTempOperState : DINT;	//Capture the Temporary Operating State of the Equipment for comparison
	
	GVL_EquipmentArray items used for Equipment Status processing
	// System Equipment
	SystemEquip_Count : INT; //Count of Equipment to Process in System PLC
	SystemEquipStatusArray : ARRAY[1..EQUIP_COUNT_MAX] OF ST_StateCntrlSts; //Array of Equipment Status Current
	SystemEquipStatusArray_Last : ARRAY[1..EQUIP_COUNT_MAX] OF ST_StateCntrlSts; //Array of Equipment Status Last State
*)

//===================================================================================
(* 	Process the Conveyor/Equipment status arrays comparing the current state to the last state
 	When a state change is deteted, add the correspoding equipment to the Msg_EquipStatArray
		Then increment/test the nEquipStatusIndex and add the message to the outbound buffer
		if the Msg_EquipStatArry is full, and reset the nEquipStatusIndex value to the lower bound
*)
// Initialise the nEquipStatusIndex to 0 to detect when items are in the Msg_EquipStatArry buffer
nEquipStatusIndex := 0;

FOR nSystemStatusIndex := 1 TO gvl_equiparrays.nSystemEquip_Count BY 1 DO
	// Test for a valid label, ignore if there isn't a label
	IF GVL_EquipArrays.aSystemEquipStatusArray[nSystemStatusIndex].Label <> '' THEN
		// Capture Offline State
		IF GVL_EquipArrays.aSystemEquipStatusArray[nSystemStatusIndex].CrntState = E_StateCntrl.stOffline THEN
			nTempOperState := E_OperStateCntrl.Offline;
		ELSE
			// Check for OverHeight
			// Initialise the stop register with the conveyor stop register
			fb_CheckStopRegister(aCodeRegister := GVL_EquipArrays.aSystemEquipStatusArray[nSystemStatusIndex].stsStopRegister);
			// Check for an OverHeight in the Stop Register
			fb_CheckStopRegister.Check(nCodeToCheck := E_StopCodes.OverHeightFLT,
				bCodeSet => bOverHeight);
			// Set over Height
			IF bOverHeight THEN
				nTempOperState := E_OperStateCntrl.OverHeight;
			ELSE
				// Capture Faulted State, or a specific Fault (in this instance, OverHeight)
				IF GVL_EquipArrays.aSystemEquipStatusArray[nSystemStatusIndex].CrntState = E_StateCntrl.stFaulted THEN
						nTempOperState := E_OperStateCntrl.Faulted;
				ELSE
					// Capture Auto/Manual States and Running/Sleeping states where appropriate
					IF GVL_EquipArrays.aSystemEquipStatusArray[nSystemStatusIndex].CrntState = E_StateCntrl.stAuto THEN
						// Capture Auto-Running
						IF GVL_EquipArrays.aSystemEquipStatusArray[nSystemStatusIndex].CrntOperState = E_OperStateCntrl.running THEN
							nTempOperState := E_OperStateCntrl.running;
						// Capture Auto-Sleeping
						ELSIF GVL_EquipArrays.aSystemEquipStatusArray[nSystemStatusIndex].CrntOperState = E_OperStateCntrl.sleeping THEN
							nTempOperState := E_OperStateCntrl.sleeping;
						// Capture Auto
						ELSE
							nTempOperState := E_OperStateCntrl.Auto;
						END_IF
					ELSE
						// Capture Manual-Running
						IF GVL_EquipArrays.aSystemEquipStatusArray[nSystemStatusIndex].CrntOperState = E_OperStateCntrl.running THEN
							nTempOperState := E_OperStateCntrl.running;
						// Capture Manual
						ELSE
							nTempOperState := E_OperStateCntrl.Manual;
						END_IF
					END_IF
				END_IF
			END_IF
		END_IF
		// Test for a change in Operational state or a non-initialized Storage array
		IF GVL_EquipArrays.aSystemEquipStatusArray_last[nSystemStatusIndex].LstOperState <> nTempOperState OR GVL_EquipArrays.aSystemEquipStatusArray_last[nSystemStatusIndex].Index = 0 THEN
			IF GVL_EquipArrays.aSystemEquipStatusArray_last[nSystemStatusIndex].Index = 0 THEN
				// Initialise the Storage Data Record
				GVL_EquipArrays.aSystemEquipStatusArray_last[nSystemStatusIndex] := GVL_EquipArrays.aSystemEquipStatusArray[nSystemStatusIndex];
			END_IF
			// Capture the nTempOperState for future comparisons
			GVL_EquipArrays.aSystemEquipStatusArray_last[nSystemStatusIndex].LstOperState := TO_INT(nTempOperState);
			// Increment the status index and check for roll-over
			nEquipStatusIndex := nEquipStatusIndex + 1;
			IF nEquipStatusIndex > 7 THEN
				// When there are 7 status updates, create the message
				TransmitMsgBuffer[TransmitMsgBuffer_Index] := EquipStatUpdate(Msg_EquipStatArry);
				// Increment the buffer index
				TransmitMsgBuffer_Index := IncIndex(TransmitMsgBuffer_Index,1,TransmitMsgBuffer_Size);
				// Set the index for the next message
				nEquipStatusIndex := 1;
			END_IF
			// Capture the Label and Index of the current Equipment status record
			Msg_EquipStatArry[nEquipStatusIndex].DeviceID := GVL_EquipArrays.aSystemEquipStatusArray[nSystemStatusIndex].Label;
			Msg_EquipStatArry[nEquipStatusIndex].Status := TO_INT(nTempOperState);
		END_IF
	END_IF
END_FOR

// Detect unsent items in the Msg_EquipStatArry buffer
IF nEquipStatusIndex > 0 THEN
	// Prepare the Equipment Status Message
	TransmitMsgBuffer[TransmitMsgBuffer_Index] := EquipStatUpdate(Msg_EquipStatArry);
	// Add the Equipment Status Message to the outbound buffer
	TransmitMsgBuffer_Index := IncIndex(TransmitMsgBuffer_Index,1,TransmitMsgBuffer_Size);
END_IF
END_ACTION

METHOD PRIVATE EquipStatUpdate : STRING(55)
VAR_IN_OUT
	Msg_ConveyorStatArry:	ARRAY[1..7] OF ST_Msg_EquipStat; // Array of Device status
END_VAR
VAR
	String1: STRING(55);
	x: INT;
	String_DefDest: STRING(2);
	y: INT;
	String_Status: STRING(2);
	Device_Len: INT;
	i: INT;
END_VAR
(* Message from communication Spec:
	[STX (0x02h)][28][Device 1 ID (5 CHR)][Status (2 CHR)] repeated for devices thru 7[ETX 0x03h)]
*)

// Start Message with header
String1 := '$0228';

FOR x := 1 TO 7 DO
	IF (Msg_ConveyorStatArry[x].DeviceID <> '') THEN
		// Check Device for length and Pad with spaces if needed
		Device_Len := LEN(Msg_ConveyorStatArry[x].DeviceID);
		IF Device_Len = 5 THEN
			String1 := CONCAT(String1,Msg_ConveyorStatArry[x].DeviceID);
		ELSIF Device_Len < 5 THEN
			Device_Len := LEN(Msg_ConveyorStatArry[x].DeviceID);
			FOR i := 1 TO (5-Device_Len) DO
				String1 := CONCAT(String1,' ');
			END_FOR
		ELSE
			String1 := CONCAT(String1, 'XXXXX');
		END_IF
		// Clear the DeviceID after processing
		Msg_ConveyorStatArry[x].DeviceID := '';
		
	
		// Check Status for length and Pad with spaces if needed
		String_Status := INT_TO_STRING(Msg_ConveyorStatArry[x].Status);
		IF Msg_ConveyorStatArry[x].Status < 10 THEN
			String1 := CONCAT(String1,'0');
			String1 := CONCAT(String1, String_Status);
		ELSIF (Msg_ConveyorStatArry[x].Status >= 10) AND (Msg_ConveyorStatArry[x].Status < 100) THEN
			String1 := CONCAT(String1, String_Status);
		ELSE
			String1 := CONCAT(String1, 'XX');
		END_IF	
		// Clear the Status after processing
		Msg_ConveyorStatArry[x].Status := 0;
	ELSE 
		String1 := CONCAT(String1,'       ');
	END_IF	
END_FOR

// Add ending Character
String1 := CONCAT(String1,'$03');
	
EquipStatUpdate := String1;
END_METHOD

METHOD PRIVATE KeepAliveResponse : STRING(55)
VAR_INPUT
END_VAR
VAR
	String1: STRING(55);
	x: INT;
END_VAR
(* Message from communication Spec:
	[STX (0x02h)][29][Blank (49 CHR)][ETX 0x03h)]
*)

// Start Message with header
String1 := '$0229';

// Pad with Spaces
FOR x := 1 TO 49 DO
	String1 := CONCAT(String1,' ');
END_FOR

// Add ending Character
String1 := CONCAT(String1,'$03');
	
KeepAliveResponse := String1;
END_METHOD

METHOD PRIVATE LocationUpdate : STRING(55)
VAR_INPUT
	Device :	STRING(5);		// Device Label per communication standard
	BarCode:	STRING(30);		// Barcode from barcode reader
	Dest:	INT;		// Default destination
END_VAR
VAR
	String1: STRING(55);
	BC_Len: INT;
	x: INT;
	String_Dest: STRING(2);
	y: INT;
	Device_Len: INT;
	i: INT;
END_VAR
(* Message from communication Spec:
	[STX (0x02h)][27][Device ID (5 CHR)][Barcode (20 CHR)][Destination (2 CHR)][Blank (24 CHR)][ETX 0x03h)]
*)

// Start Message with header
String1 := '$0227';

// Check Device for length and Pad with spaces if needed
Device_Len := LEN(Device);
IF Device_Len = 5 THEN
	String1 := CONCAT(STRING1, Device);
ELSIF Device_Len < 5 THEN
	String1 := CONCAT(STRING1, Device);
	FOR i := 1 TO (5-Device_Len) DO
		String1 := CONCAT(String1,' ');
	END_FOR	
ELSE
	String1 := CONCAT(String1, 'XXXXX');
END_IF


// Check Barcode for length and Pad with spaces if needed
BC_Len := LEN(BARCODE);
IF BC_Len <20 THEN
	String1 := CONCAT(STRING1, BarCode);
	FOR x := 1 TO (20-BC_Len) DO
		String1 := CONCAT(String1,' ');
	END_FOR
ELSIF BC_Len = 20 THEN
	String1 := CONCAT(STRING1, BarCode);
ELSE 
	String1 := CONCAT(STRING1, RIGHT(BarCode,20));	
END_IF

(* Destination isn't needed in location Update 
// Check Default Destination for length and Pad with spaces if needed
String_Dest := INT_TO_STRING(Dest);
IF Dest < 10 THEN
	String1 := CONCAT(String1,'0');
	String1 := CONCAT(String1, String_Dest);
ELSIF (Dest >= 10) AND (Dest < 100) THEN
	String1 := CONCAT(String1, String_Dest);
ELSE
	String1 := CONCAT(String1, 'XX');
END_IF	
*)

// Pad with spaces
FOR y := 1 TO 24 DO
	String1 := CONCAT(String1,' ');
END_FOR

// Add ending Character
String1 := CONCAT(String1,'$03');
	
LocationUpdate := String1;
END_METHOD

ACTION RECEIVE:
// Empty all outputs
	DeviceID := BarCode := '';
	Destination := DefDestination := 0;
	Status := 99;
	Msg_EquipStatArry := Blank_Msg_ConveyorStatArry;

	// Set up index with clipping to keep it within array boundaries	
	i := IncIndex(i,1,10);
		
	// Clear one before to make it easy to find newest entry 
	IF i = 10 THEN
		RawMsgArray[1] := '';	
		RawMsgLenArray[1] := 0;	
		RawMsgStartPosArray[1] := 0;
		RawMsgEndPosArray[1] :=  0;
	ELSE
		RawMsgArray[i+1] := '';	
		RawMsgLenArray[i+1] := 0;	
		RawMsgStartPosArray[i+1] := 0;
		RawMsgEndPosArray[i+1] :=  0;
	END_IF
	
	
	// Fill Appropriate info for each message
	RawMsgArray[i] := ServerControl.fbServer.aApplications[nConnectionIndex].RxRawMessage;	
	RawMsgLenArray[i] := LEN(ServerControl.fbServer.aApplications[nConnectionIndex].RxRawMessage);	
	StrStartPos := FIND(STR1:= RawMsgArray[i], STR2:='$02' );
	StrEndPos :=  FIND(STR1:= RawMsgArray[i], STR2:='$03' );
	RawMsgStartPosArray[i] := StrStartPos;
	RawMsgEndPosArray[i] := StrEndPos;
	
{info 'Maybe: Possibly add do while loop here to process the case where more than one message comes in at a time and clean up StrStartPos and end pos with array'}	
	IF StrStartPos <> 0 THEN
		MsgString := MID(STR:=ServerControl.fbServer.aApplications[nConnectionIndex].RxRawMessage , LEN:= 51 , POS:= StrStartPos);
		MsgArray[i] := MsgString;
		MsgID := STRING_TO_DINT(MID(STR:=ServerControl.fbServer.aApplications[nConnectionIndex].RxRawMessage , LEN:= 2, POS:= StrStartPos+1));
	
		CASE MsgID OF
			E_MessageIds.TransportCommand_05:  	// Transport Command Message
				DeviceID := MID(STR:=ServerControl.fbServer.aApplications[nConnectionIndex].RxRawMessage, LEN:= 5, POS:= StrStartPos+3);
				BarCode := MID(STR:=ServerControl.fbServer.aApplications[nConnectionIndex].RxRawMessage, LEN:= 20, POS:= StrStartPos+8);
				Destination := STRING_TO_DINT( MID(STR:=ServerControl.fbServer.aApplications[nConnectionIndex].RxRawMessage, LEN:= 2, POS:= StrStartPos+28));
				DefDestination := STRING_TO_DINT( MID(STR:=ServerControl.fbServer.aApplications[nConnectionIndex].RxRawMessage, LEN:= 2, POS:= StrStartPos+30));
				Status := STRING_TO_BYTE( MID(STR:=ServerControl.fbServer.aApplications[nConnectionIndex].RxRawMessage , LEN:= 2, POS:= StrStartPos+50));

				//Strip spaces from Bar Code
				SpacePosition := (FIND(STR1:= BarCode, STR2:=' ' ))+3;
				BarCodeNoSpace := MID(STR:=BarCode, LEN:= (20-SpacePosition), POS:= 1);
				// Update Info to send to Sorter PLC
//				ItemTransport := BlankItem;
				ItemTransport.DeviceID := DeviceID;
				ItemTransport.ID := BarCodeNoSpace;
				ItemTransport.Destination := Destination;
				ItemTransport.Status := E_StatusCode.UpdateNeeded;
				ItemTransport.MessageType := E_MessageIds.TransportCommand_05;
//				fb_SorterTransportBuffer.AddItem(st_ItemToAdd := ItemTransport);
//				Out_DefaultDestination := DefDestination;

			E_MessageIds.LocationUpdateResponse_07:		// Location Update Response
				DeviceID := MID(STR:=ServerControl.fbServer.aApplications[nConnectionIndex].RxRawMessage , LEN:= 5, POS:= StrStartPos+3);
				BarCode := MID(STR:=ServerControl.fbServer.aApplications[nConnectionIndex].RxRawMessage , LEN:= 20, POS:= StrStartPos+8);
				Destination := STRING_TO_DINT( MID(STR:=ServerControl.fbServer.aApplications[nConnectionIndex].RxRawMessage , LEN:= 2, POS:= StrStartPos+23));
				Status := STRING_TO_BYTE( MID(STR:=ServerControl.fbServer.aApplications[nConnectionIndex].RxRawMessage , LEN:= 2, POS:= StrStartPos+50));
						
			E_MessageIds.EquipmentStatusResponse_08:		// Equipment Status Response
				FOR j := 0 TO 6 DO
					Msg_EquipStatArry[j+1].DeviceID := MID(STR:=ServerControl.fbServer.aApplications[nConnectionIndex].RxRawMessage , LEN:= 5, POS:= ((StrStartPos+3)+(j*7)));
					Msg_EquipStatArry[j+1].Status := STRING_TO_BYTE(MID(STR:=ServerControl.fbServer.aApplications[nConnectionIndex].RxRawMessage , LEN:= 2, POS:= ((StrStartPos+8)+(j*7))));	
				END_FOR
			
			E_MessageIds.KeepAlive_09:		// Keep Alive
				// If Keep Alive message is recieved send the response to the transmit buffer
				TransmitMsgBuffer[TransmitMsgBuffer_Index] := KeepAliveResponse();
				TransmitMsgBuffer_Index := IncIndex(TransmitMsgBuffer_Index,1,TransmitMsgBuffer_Size);				
		END_CASE
	END_IF
END_ACTION

ACTION TRANSMIT:

// Transmit messages from buffer
IF NOT ServerControl.TransmitTrigger AND TransmitEnable THEN
	ServerControl.TxMessage := TransmitMsgBuffer[SendingMsg_Index];
	ServerControl.TransmitTrigger := TRUE;
	SendingMsg_Index := IncIndex(SendingMsg_Index,1,TransmitMsgBuffer_Size);
	
	TransmittedArray[y] := ServerControl.TxMessage;
	// Clear out message before last update to ease in testing
	IF y = 10 THEN
		TransmittedArray[1] := '';
	ELSE
		TransmittedArray[y+1] := '';
	END_IF
	
	y :=  IncIndex(IDX:= y, IdxMIN:= 0, IdxMAX:=10 );
END_IF
END_ACTION

METHOD PRIVATE TransportComplete : STRING(55)
VAR_INPUT
	Device :	STRING(5);		// Device Label per communication standard
	BarCode:	STRING(30);		// Barcode from barcode reader
	Dest:	INT;		// Default destination
	Status:	INT;		// Status
END_VAR
VAR
	String1: STRING(55);
	BC_Len: INT;
	x: INT;
	String_Dest: STRING(2);
	y: INT;
	String_Status: STRING(2);
	Device_Len: INT;
	i: INT;
END_VAR
(* Message from communication Spec:
	[STX (0x02h)][26][Device ID (5 CHR)][Barcode (20 CHR)][Destination (2 CHR)][Blank (20 CHR)][Status (2 CHR)][ETX 0x03h)]
*)

// Start Message with header
String1 := '$0226';

// Check Device for length and Pad with spaces if needed
Device_Len := LEN(Device);
IF Device_Len = 5 THEN
	String1 := CONCAT(STRING1, Device);
ELSIF Device_Len < 5 THEN
	String1 := CONCAT(STRING1, Device);
	FOR i := 1 TO (5-Device_Len) DO
		String1 := CONCAT(String1,' ');
	END_FOR
ELSE
	String1 := CONCAT(String1, 'XXXXX');
END_IF

// Check Barcode for length and Pad with spaces if needed
BC_Len := LEN(BARCODE);
IF BC_Len <20 THEN
	String1 := CONCAT(STRING1, BarCode);
	FOR x := 1 TO (20-BC_Len) DO
		String1 := CONCAT(String1,' ');
	END_FOR
ELSIF BC_Len = 20 THEN
	String1 := CONCAT(STRING1, BarCode);
ELSE 
	String1 := CONCAT(STRING1, RIGHT(BarCode,20));	
END_IF

// Check Destination for length and Pad with spaces if needed
String_Dest := INT_TO_STRING(Dest);
IF Dest < 10 THEN
	String1 := CONCAT(String1,'0');
	String1 := CONCAT(String1, String_Dest);
ELSIF (Dest >= 10) AND (Dest < 100) THEN
	String1 := CONCAT(String1, String_Dest);
ELSE
	String1 := CONCAT(String1, 'XX');
END_IF	

// Pad with Spaces
FOR y := 1 TO 20 DO
	String1 := CONCAT(String1,' ');
END_FOR

// Check Status for length and Pad with spaces if needed
String_Status := INT_TO_STRING(Status);
IF Status < 10 THEN
	String1 := CONCAT(String1,'0');
	String1 := CONCAT(String1, String_Status);
ELSIF (Status >= 10) AND (Status < 100) THEN
	String1 := CONCAT(String1, String_Status);
ELSE
	String1 := CONCAT(String1, 'XX');
END_IF	

// Add ending Character
String1 := CONCAT(String1,'$03');
	
TransportComplete := String1;
END_METHOD

METHOD PRIVATE TransportResponse : STRING(55)
VAR_INPUT
	Device :	STRING(5);		// Device Label per communication standard
	BarCode :	STRING(30);		// Barcode from barcode reader
	Status :	INT;		// Status
END_VAR
VAR
	String1: STRING(55);
	BC_Len: INT;
	x: INT;
	String_Status: STRING(2);
	y: INT;
	Device_Len: INT;
	i: INT;
END_VAR
(* Message from communication Spec:
	[STX (0x02h)][25][Device ID (5 CHR)][Barcode (20 CHR)][Blank (22 CHR)][Status (2 CHR)][ETX 0x03h)]
*)

// Start Message with header
String1 := '$0225';

// Check Device for length and Pad with spaces if needed
Device_Len := LEN(Device);
IF Device_Len = 5 THEN
	String1 := CONCAT(STRING1, Device);
ELSIF Device_Len < 5 THEN
	String1 := CONCAT(STRING1, Device);
	FOR i := 1 TO (5-Device_Len) DO
		String1 := CONCAT(String1,' ');
	END_FOR
ELSE
	String1 := CONCAT(String1, 'XXXXX');
END_IF

// Check Barcode for length and Pad with spaces if needed
BC_Len := LEN(BARCODE);
IF BC_Len <20 THEN
	String1 := CONCAT(STRING1, BarCode);
	FOR x := 1 TO (20-BC_Len) DO
		String1 := CONCAT(String1,' ');
	END_FOR
ELSIF BC_Len = 20 THEN
	String1 := CONCAT(STRING1, BarCode);
ELSE 
	String1 := CONCAT(STRING1, RIGHT(BarCode,20));	
END_IF

// Pad with Spaces
FOR y := 1 TO 22 DO
	String1 := CONCAT(String1,' ');
END_FOR

// Check Status for length and Pad with spaces if needed
String_Status := INT_TO_STRING(Status);
IF Status < 10 THEN
	String1 := CONCAT(String1,'0');
	String1 := CONCAT(String1, String_Status);
ELSIF (Status >= 10) AND (Status < 100) THEN
	String1 := CONCAT(String1, String_Status);
ELSE
	String1 := CONCAT(String1, 'XX');
END_IF

// Add ending Character
String1 := CONCAT(String1,'$03');
	
TransportResponse := String1;
END_METHOD

END_PROGRAM

// ---- POUs/ServerControl.TcPOU
PROGRAM ServerControl
VAR_INPUT
	TxMessage			: 	STRING(55);
	TransmitTrigger 	: 	BOOL;
END_VAR
VAR
	{attribute 'OPC.UA.DA' := '1'}
	bInitialize			: 	BOOL := TRUE;

	nIndexInit			:	UDINT;
	nCurrentServerIndex	:	UDINT := 1;			// Index of the currently communicating server, initialize to the first server instance

	sSrvNetID			: 	T_AmsNetID	:= '';		// TwinCAT TCP/IP server AMS network address
	fbServer			: 	FB_Server ;
	fbCloseAll			: 	FB_SocketCloseAll;
	aTransmitTrigger	: 	ARRAY [1..ServerControl.MAX_CLIENT_CONNECTIONS] OF BOOL;
	{attribute 'OPC.UA.DA' := '1'}
	aEnable				: 	ARRAY [1..ServerControl.MAX_CLIENT_CONNECTIONS] OF BOOL;			// TRUE => Enable server data exchange, FALSE => Disable
	aLog				: 	ARRAY [1..ServerControl.MAX_CLIENT_CONNECTIONS] OF BOOL;					// TRUE => Enable message/error log, FALSE => Disable
END_VAR

VAR CONSTANT	
	MAX_CLIENT_CONNECTIONS					: UDINT(1..20) := 1;	// Possible number of client connections
	PLCPRJ_BUFFER_SIZE						: UDINT := 1000;		// Max. internal fifo/receiver buffer size
	PLCPRJ_RECEIVE_POLLING_TIME				: TIME := T#100MS;
	PLCPRJ_RECEIVE_TIMEOUT					: TIME := T#15M;		// Timeout if no data is received

	// Project specific error codes
	PLCPRJ_ERROR_RECEIVE_TIMEOUT			: UDINT := 16#8101;		// Receive timeout
	PLCPRJ_ERROR_SENDFIFO_OVERFLOW			: UDINT := 16#8102;		// Send fifo overflow
	PLCPRJ_ERROR_RECFIFO_OVERFLOW			: UDINT := 16#8103;		// Receive fifo overflow
END_VAR

(* On PLC reset or program download close all created/opened sockets/connections *)
fbCloseAll( sSrvNetID := sSrvNetID, bExecute:= bInitialize );
IF fbCloseAll.bBusy OR fbCloseAll.bError THEN
	RETURN;
END_IF

IF bInitialize then
	// Setup Server data, Own IP, communicating port, logging prefix
	fbServer.sLocalHost := '0.0.0.0';
	fbServer.nLocalPort := 49200;
	fbServer.sPrefix := 'SERVER::';
end_if

bInitialize := FALSE;

// Allow the logs to be turned on/off
// And set the Server enables
// Filter by nIndexInit to disable/enable specific Server instances
FOR nIndexInit:= 1 TO MAX_CLIENT_CONNECTIONS DO
	aLog[nIndexInit] := .nServerLogEnable.BUFFER_LOG;
	aEnable[nIndexInit] := TRUE;
END_FOR

// Identify the trigger to use for sending
aTransmitTrigger[nCurrentServerIndex] := TransmitTrigger;

// Call the server block
fbServer( TxMessage := TxMessage, aTransmitTrigger := aTransmitTrigger, sSrvNetID := sSrvNetID, aEnable := aEnable, aLog := aLog
		, nServerIndex => nCurrentServerIndex);

MsgControl(nConnectionIndex := nCurrentServerIndex);		// Control the messages being sent out via TCP/IP

END_PROGRAM

// ---- FunctionBlocks/Server/FB_Server.TcPOU
FUNCTION_BLOCK FB_Server
VAR_INPUT
	sSrvNetID			: 	T_AmsNetID	:= '';			(* TwinCAT TCP/IP server network address *)
	sLocalHost			: 	T_IPv4Addr 	:= '0.0.0.0';	(* Own IP address!, all Zeros if server *)
	nLocalPort			: 	UDINT 		:= 0;			(* Server port number *)
	tReconnect 			: 	TIME 		:= T#3S;		(* Reopen new listener socket after this time *)
	sPrefix				: 	STRING 		:= 'SERVER::';	(* Log message description string (allows the identification of log message source) *)
	aTransmitTrigger	: 	ARRAY[1..ServerControl.MAX_CLIENT_CONNECTIONS] OF BOOL;
	aEnable				:	ARRAY[1..ServerControl.MAX_CLIENT_CONNECTIONS] OF BOOL;		(* TRUE => enable server data exchange, FALSE => disable *)
	aLog				: 	ARRAY[1..ServerControl.MAX_CLIENT_CONNECTIONS] OF BOOL;		(* TRUE => Enable log message output, FALSE => Disable *)
	TxMessage			: 	STRING(55);
	bEnable				:	BOOL;
	bLog				:	BOOL;
END_VAR

VAR_OUTPUT
	{attribute 'OPC.UA.DA' := '1'}
	bListening		: BOOL			:= FALSE;(* Listener socket state *)
	{attribute 'OPC.UA.DA' := '1'}
	nAccepted		: UDINT			:= 0;(* Number of accepted client connections *)
	{attribute 'OPC.UA.DA' := '1'}
	nServerIndex	: UDINT			:= 1;(* Index of Currently communicating Server, initialize to the first server *)
END_VAR
VAR
	aApplications	: ARRAY[1..ServerControl.MAX_CLIENT_CONNECTIONS] OF FB_ServerApplication;(* Server application control function blocks *)
	aConnections	: ARRAY[1..ServerControl.MAX_CLIENT_CONNECTIONS] OF FB_ServerConnection;(* Server connection/data exchange control function blocks *)
	aTx 			: ARRAY[1..ServerControl.MAX_CLIENT_CONNECTIONS] OF FB_FrameFifo;(* TX fifo *)
	aRx 			: ARRAY[1..ServerControl.MAX_CLIENT_CONNECTIONS] OF FB_FrameFifo;(* RX fifo *)
	aLogFifo		: ARRAY[1..ServerControl.MAX_CLIENT_CONNECTIONS] OF FB_LogFifo;(* Listener log message fifo *)
	fbListen	 	: FB_SocketListen;
	fbClose			: FB_SocketClose;
	fbLog			: FB_LogFifo;
	fbListenTimer	: TON;
	{attribute 'OPC.UA.DA' := '1'}
	bReset			: BOOL := FALSE;
	bConnecting		: BOOL;
	eStep			: E_ServerSteps;
	i				: UDINT;
END_VAR

// Set to FALSE each time this is run
bEnable := FALSE; 
// Test for any enabled connections
FOR i:= 1 TO ServerControl.MAX_CLIENT_CONNECTIONS DO
	IF aEnable[i] THEN
		bEnable := TRUE; 
	END_IF
END_FOR

// Set to FALSE each time this is run
bLog := FALSE; 
// Test for any enabled connections
FOR i:= 1 TO ServerControl.MAX_CLIENT_CONNECTIONS DO
	IF aLog[i] THEN
		bLog := TRUE; 
	END_IF
END_FOR

// Test the current State of the Listening Socket
CASE eStep OF
	(*
		Idle connections can transition to 
			LISTENER_OPEN_START
			REMOTE_CLIENTS_CLOSE
			REMOTE_CLIENTS_COMM
	*)
	eSERVER_STATE_IDLE:
		// If Listening and not enabled, Set REMOTE_CLIENTS_CLOSE
		// Otherwise, set LISTENING_OPEN_START after the listen timer expires
		IF bEnable XOR bListening THEN
			IF bEnable THEN
				fbListenTimer( IN := TRUE );
				IF fbListenTimer.Q THEN
					fbListenTimer( IN := FALSE, PT := tReconnect );

					fbLog.Clear( sPrefix := sPrefix, bLog := bLog );(* Clear listener log fifo *)
					bReset := FALSE;

					eStep := eSERVER_STATE_LISTENER_OPEN_START;
				END_IF
			ELSE
				eStep := eSERVER_STATE_REMOTE_CLIENTS_CLOSE;
			END_IF
		ELSIF bListening THEN
			eStep := eSERVER_STATE_REMOTE_CLIENTS_COMM;
		ELSE
			fbListenTimer( IN := FALSE, PT := T#0S );
			bReset := FALSE;
		END_IF

	(*
		LISTENER_OPEN_START transitions to LISTENER_OPEN_WAIT
	*)
	eSERVER_STATE_LISTENER_OPEN_START:
		// FB_SocketListen executes on the leading edge or bExecute, so setting it to false then true causes it to listen
		fbListen(  bExecute := FALSE  );
		fbListen( 	sSrvNetID := sSrvNetID, 
					sLocalHost := sLocalHost, 
					nLocalPort := nLocalPort, 
					bExecute := TRUE );
		eStep := eSERVER_STATE_LISTENER_OPEN_WAIT;

	(*
		LISTENER_OPEN_START transitions to IDLE or ERROR, depending on the results of the FB_SocketListen call
		When the results are good, bListening is set to TRUE and the server state is IDLE
		When an error occurs, the ERROR state is initiated
	*)
	eSERVER_STATE_LISTENER_OPEN_WAIT:
		fbListen( bExecute := FALSE );
		IF NOT fbListen.bBusy THEN
			IF NOT fbListen.bError THEN
				bListening 	:= TRUE;
				fbLog.Message( sMessage := 'Listener socket opened!', hSocket := fbListen.hListener );
				eStep := eSERVER_STATE_IDLE;
			ELSE
				fbLog.Error( sMessage := 'FB_SocketListen()', nErrId := fbListen.nErrId );
				eStep := eSERVER_STATE_ERROR;
			END_IF
		END_IF

	(*
		REMOTE_CLIENTS_COMM transitions to IDLE ot REMOTE_CLIENTS_CLOSE depending on the state of the bReset signal
	*)
	eSERVER_STATE_REMOTE_CLIENTS_COMM:
		eStep := eSERVER_STATE_IDLE;
		nAccepted := 0;
		bConnecting := FALSE;

		FOR i:= 1 TO ServerControl.MAX_CLIENT_CONNECTIONS DO
			aConnections[i].sPrefix := CONCAT(CONCAT('SERVER',UDINT_TO_STRING(i)),'::');
			aConnections[i](bAllowConnect := NOT bConnecting
							, fbTx := aTx[i], fbRx := aRx[i], fbLog := aLogFifo[i]
							, hListener := fbListen.hListener, bReset := bReset
							, sSrvNetID := sSrvNetID, bEnable := aEnable[i],	bLog := aLog[i] 
							, bConnecting=>bConnecting); 
			IF bReset THEN
				bReset := FALSE; 
				eStep := eSERVER_STATE_REMOTE_CLIENTS_CLOSE;
				EXIT;
			END_IF
			
			nServerIndex := 1;
			IF aConnections[i].bAccepted OR aTransmitTrigger[i] THEN  // OR aTransmitTrigger[i] Clear send message even if no connection is made
				aApplications[i]( TxMessage := TxMessage
								, bTransmitTrigger := aTransmitTrigger[i]
								, fbTx := aTx[i]
								, fbRx := aRx[i]
								, fbLog := aLogFifo[i] );
				// Adjust the server index to the last accepted connection
				IF nServerIndex <> i THEN
					nServerIndex := i;
				END_IF
				nAccepted := nAccepted + 1;(* Count the number of connected remote clients *)
			END_IF

		END_FOR

	(*
		REMOTE_CLIENTS_CLOSE transitions to LISTENER_CLOSE_START
		First all enabled connections are set to FALSE to close them.
		The server remains in this state until all connections are closed
		It then transitions to LISTENER_CLOSE_START to close the listening socket
	*)
	eSERVER_STATE_REMOTE_CLIENTS_CLOSE:
		nAccepted := 0;
		FOR i:= 1 TO ServerControl.MAX_CLIENT_CONNECTIONS DO
			(* Close all remote client (accepted) sockets *)
			aConnections[i]( fbTx := aTx[i], fbRx := aRx[i], fbLog := aLogFifo[i],
							hListener := fbListen.hListener, bReset := bReset,
							sSrvNetID := sSrvNetID, bEnable := FALSE, bLog := aLog[i] ); 
			IF aConnections[i].bAccepted THEN
				nAccepted := nAccepted + 1;(* Count the number of connected remote clients *)
			END_IF
		END_FOR
		
		(* Check if all remote client sockets are closed *)
		IF nAccepted = 0 THEN
			eStep := eSERVER_STATE_LISTENER_CLOSE_START; (* Close listener socket too *)
		END_IF

	(*
		LISTENER_CLOSE_START transitions to LISTENER_CLOSE_WAIT after the FB_SocketClose function block is called
	*)
	eSERVER_STATE_LISTENER_CLOSE_START:
		fbLog.Message( sMessage := 'Closing listener socket!', hSocket := fbListen.hListener );
		fbClose( bExecute := FALSE );
		fbClose( sSrvNetID := sSrvNetID, hSocket := fbListen.hListener, bExecute:= TRUE );
		eStep := eSERVER_STATE_LISTENER_CLOSE_WAIT;

	(*
		LISTENER_CLOSE_WAIT transitions to IDLE or ERROR dependig on the result of the FB_CloseSocket call
	*)
	eSERVER_STATE_LISTENER_CLOSE_WAIT:
		fbClose( bExecute := FALSE );
		IF NOT fbClose.bBusy THEN
			bListening := FALSE;
			nAccepted := 0;
			IF NOT fbClose.bError THEN
				eStep := eSERVER_STATE_IDLE;
			ELSE
				fbLog.Error( sMessage := 'FB_SocketClose(listener)', nErrId := fbListen.nErrID );
				eStep := eSERVER_STATE_ERROR;
			END_IF
		END_IF

	(*
		LISTENER_OPEN_START transitions to IDLE or REMOTE_CLIENTS_CLOSE, depending on the state of the listening socket
		When not listening the server state is set to IDLE
		When listening, the state is set to REMOTE_CLIENTS_CLOSE
	*)
	eSERVER_STATE_ERROR:
		IF bListening THEN
			eStep := eSERVER_STATE_REMOTE_CLIENTS_CLOSE;
		ELSE
			eStep := eSERVER_STATE_IDLE;
		END_IF

END_CASE

END_FUNCTION_BLOCK

// ---- FunctionBlocks/Server/FB_ServerApplication.TcPOU
FUNCTION_BLOCK FB_ServerApplication
VAR_INPUT
	TxMessage :	STRING(55);		// Message to Transmit
	bTransmitTrigger: BOOL;		// Trigger to add TxMessage to the TCP/IP send Buffer (TRUE= Trasmit On Rising Edge Only)
END_VAR
VAR_IN_OUT
	fbTx 		: FB_FrameFifo;(* TX fifo *)
	fbRx 		: FB_FrameFifo;(* RX fifo *)
	fbLog		: FB_LogFifo;(* Log message fifo *)
END_VAR
VAR_OUTPUT
	TxCounter	: UDINT;	// Shows that the transmit message was added to the transmt buffer 
	RxCounter	: UDINT;	// Shows that a message was recieved
	RxRawMessage: STRING(255);		// Message output
END_VAR
VAR
	sToClient	: T_MaxString := '';
	sFromClient	: T_MaxString := '';
	sLogMessage	: T_MaxString := '';
	TxTrigger: R_TRIG;
END_VAR

(*------------------- Send message strings ------------------------------------*)
// TxTrigger(CLK:= bTransmitTrigger);

IF (* TxTrigger.Q*) bTransmitTrigger  THEN(* Send string to server *)
	
	sToClient := TxMessage; // Message
 		
	fbTx.AddTail( sPut := sToClient );(* Put string to the tx fifo *)
	IF NOT fbTx.bOk THEN(* TX fifo overflow => log error *)
		fbLog.Error( sMessage := 'FB_FrameFifo(sender)', nErrID := ServerControl.PLCPRJ_ERROR_SENDFIFO_OVERFLOW );
	END_IF
	
	TxCounter := TxCounter  + 1;
	// bTransmitTrigger := FALSE;
END_IF

(*------------------------------- Get received message strings ---------------------------------*)
REPEAT
	fbRx.RemoveHead( );(* Fetch string from rx fifo *)
	IF fbRx.bOk THEN(* Success *)
		
		sFromClient := fbRx.sGet;
		RxRawMessage := sFromClient;	// This could be set on line above left seperate in case some manipulation was needed before sending out
		
	(* Send back what was recieved for testing
		fbTx.AddTail( sPut := sToClient );(* Put string to the tx fifo *)
		IF NOT fbTx.bOk THEN(* TX fifo overflow => log error *)
			fbLog.Error( sMessage := 'FB_FrameFifo(sender)', nErrID := ServerControl.PLCPRJ_ERROR_SENDFIFO_OVERFLOW ); 
		END_IF
	*)
	
		RxCounter := RxCounter +1;  // Increment counter to show that data was recieved
		
		
	END_IF
UNTIL NOT fbRx.bOk
END_REPEAT

(*------------------------------- Get log/error messages from log fifo ---------------------------*)
REPEAT
	fbLog.Remove( );
	IF fbLog.bOk THEN(* Success *)
		
		(* TODO: Implement log message handler *)
		sLogMessage := fbLog.sGet;
		
	END_IF
UNTIL NOT fbLog.bOk
END_REPEAT

END_FUNCTION_BLOCK

// ---- FunctionBlocks/Server/Helper POUs/FB_FrameFifo.TcPOU
(* Tx/Rx (string data) fifo control function block *)
FUNCTION_BLOCK FB_FrameFifo
VAR_INPUT
	bLog		: BOOL			:= FALSE;(* TRUE => Enable log message output, FALSE => Disable *)
	sPrefix		: STRING		:= 'Unknown::';(* Log message description string (allows the identification of log message source) *)
	sPut		: T_MaxString 	:= ''; (* String message to add (write) to the fifo *)
END_VAR
VAR_OUTPUT
	bOk			: BOOL; 	 	(* TRUE = New entry added or removed succesfully, FALSE = Fifo overflow or fifo empty *)
	sGet		: T_MaxString 	:= '';(* String message removed (read) from fifo *)
	nCount		: UDINT			:= 0;(* Number of fifo entries *)
	cbFree		: UDINT 		:= 0;(* Free buffer space *)
	msgType		: SINT;			// Extract the message type to determine if we are logging it
	ncbSize		: UDINT;		// (*Buffer assigned bytes*)
END_VAR
VAR
	fbBuffer 	: FB_StringRingBuffer := (bOverwrite := FALSE);(* Basic (lower level) string buffer control function block *)
	buffer		: ARRAY[-3..ServerControl.PLCPRJ_BUFFER_SIZE] OF BYTE;(* Internal buffer memory *)
END_VAR

;

ACTION AddTail:
(* Adds new fifo entry *)
fbBuffer.A_AddTail( pBuffer:= ADR(buffer), cbBuffer:= SIZEOF(buffer),
					putValue:= sPut, bOk=>bOk, nCount=>nCount, cbSize=>ncbSize );

IF bOk THEN
	cbFree := ServerControl.PLCPRJ_BUFFER_SIZE - fbBuffer.cbSize;(* Calculate the free buffer space *)
	IF bLog THEN(* Log message *)
		msgType := STRING_TO_SINT(MID(sPut,2,2));
		// Ignore frequent messages
		IF (msgType = TransportCommand_05 AND nMessageLogEnable.TransportCommand_05)
		   OR (msgType = E_MessageIds.LocationUpdateResponse_07 AND nMessageLogEnable.LocationUpdateResponse_07)
		   OR (msgType = E_MessageIds.EquipmentStatusResponse_08 AND nMessageLogEnable.EquipmentStatusResponse_08)
		   OR (msgType = E_MessageIds.KeepAlive_09 AND nMessageLogEnable.KeepAlive_09)
		   OR (msgType = E_MessageIds.Arrival_23 AND nMessageLogEnable.Arrival_23)
		   OR (msgType = E_MessageIds.TransportResponse_25 AND nMessageLogEnable.TransportResponse_25)
		   OR (msgType = E_MessageIds.TransportComplete_26 AND nMessageLogEnable.TransportComplete_26)
		   OR (msgType = E_MessageIds.LocationUpdate_27 AND nMessageLogEnable.LocationUpdate_27)
		   OR (msgType = E_MessageIds.EquipmentStatusUpdate_28 AND nMessageLogEnable.EquipmentStatusUpdate_28)
		   OR (msgType = E_MessageIds.KeepAliveResponse_29 AND nMessageLogEnable.KeepAliveResponse_29)
		   OR (msgType = E_MessageIds.NoMessage_00)
		   THEN
			ADSLOGSTR( ADSLOG_MSGTYPE_HINT OR ADSLOG_MSGTYPE_LOG, CONCAT( sPrefix, '"%s"' ), sPut );
		END_IF
	END_IF
END_IF
END_ACTION

ACTION Clear:
(* Resets fifo = clears all data *)
fbBuffer.A_Reset( pBuffer:= ADR(buffer), cbBuffer:= SIZEOF(buffer),
				bOk=>bOk, getValue=>sGet, nCount=>nCount, cbSize=>ncbSize );
cbFree := ServerControl.PLCPRJ_BUFFER_SIZE;(* Free buffer size *)

sPut := CONCAT(CONCAT( sPrefix, 'Frame Buffer Cleared' ), CONCAT( CONCAT('::Queued Strings ', UDINT_TO_STRING(nCount)),CONCAT('::Used Buffer Size ', UDINT_TO_STRING(ncbSize))) );

IF bOk THEN
	IF bLog THEN(* Log information message *)
		ADSLOGSTR( ADSLOG_MSGTYPE_HINT OR ADSLOG_MSGTYPE_LOG, '%s', sPut );	
	END_IF
END_IF
END_ACTION

ACTION RemoveHead:
(* Removes oldest fifo entry *)
fbBuffer.A_RemoveHead( pBuffer:= ADR(buffer), cbBuffer:= SIZEOF(buffer),
						bOk=>bOk, getValue=>sGet, nCount=>nCount );
IF bOk THEN
	cbFree := ServerControl.PLCPRJ_BUFFER_SIZE - fbBuffer.cbSize;(* Calculate the free buffer space *)
END_IF
END_ACTION

END_FUNCTION_BLOCK

// ---- FunctionBlocks/Server/Helper POUs/FB_LogFifo.TcPOU
(* Log/debug/error message fifo *)
FUNCTION_BLOCK FB_LogFifo
VAR_INPUT
	bLog		: BOOL 		:= FALSE;(* TRUE => Enable log message output, FALSE => Disable *)
	sPrefix		: STRING 	:= 'Unknown::';(* Log message description string (allows the identification of log message source) *)
	
	sMessage	: STRING 	:= '';(* String message to add (write) to the fifo *)
	nErrID		: UDINT 	:= 0;(* Error code to add (write) to the fifo *)
	hSocket		: T_HSOCKET;(* Socket connection handle *)
END_VAR
VAR_OUTPUT
	bOk			: BOOL;(* TRUE = New entry added or removed succesfully, FALSE = Fifo overflow or fifo empty *)
	sGet		: T_MaxString := '';(* String entry removed (read) from fifo *)
	nCount		: UDINT := 0;(* Number of fifo entries *)
	ncbSize		: UDINT := 0; (* Bytes assigned to the buffer*)
END_VAR
VAR
	fbBuffer 	: FB_StringRingBuffer;(* Basic (lower level) string buffer control function block *)
	buffer		: ARRAY[0..ServerControl.PLCPRJ_BUFFER_SIZE] OF BYTE;(* Internal buffer memory *)
	sSource		: T_MaxString;	
	sPut		: T_MaxString;
END_VAR

;

ACTION Clear:
(* Clears all fifo entries *)
fbBuffer.A_Reset( 	pBuffer := ADR( buffer ), cbBuffer := SIZEOF( buffer ), 
					bOk=>bOk, nCount=>nCount, getValue=>sGet, cbSize=>ncbSize); 

sPut := CONCAT( CONCAT( sPrefix, 'Log Buffer Cleared' ), CONCAT( CONCAT('::Queued Strings ', UDINT_TO_STRING(nCount)),CONCAT('::Used Buffer Size ', UDINT_TO_STRING(ncbSize))) );

IF bOk THEN
	IF bLog THEN(* Log information message *)
		ADSLOGSTR( ADSLOG_MSGTYPE_HINT OR ADSLOG_MSGTYPE_LOG, '%s', sPut );	
	END_IF
END_IF
END_ACTION

ACTION Error:
(* Adds new fifo entry *)
IF nErrID = 0 THEN
	sSource := '::Error: 0x';
ELSIF ( nErrID AND 16#80000000) = 16#80000000 THEN
	IF nErrID = 16#80072746 THEN
		sSource := '::Win32 error (the connection is reset by remote side): 0x';
	ELSE
		sSource := '::Win32 error: 0x';
	END_IF
ELSIF (nErrID AND 16#00008100) = 16#00008100 THEN
	CASE nErrID OF
		ServerControl.PLCPRJ_ERROR_RECEIVE_TIMEOUT:
			sSource := '::PLC receive timeout error: 0x';
		ServerControl.PLCPRJ_ERROR_SENDFIFO_OVERFLOW:
			sSource := '::PLC send fifo overflow error: 0x';
		ServerControl.PLCPRJ_ERROR_RECFIFO_OVERFLOW:
			sSource := '::PLC receive fifo overflow error: 0x';
	ELSE
		sSource := '::Other PLC TCP error: 0x';
	END_CASE
ELSIF (nErrID AND 16#00008000) = 16#00008000 THEN
	sSource := '::Internal TCP/IP Connection Server error: 0x';
ELSE
	sSource := '::TwinCAT System error: 0x';
END_IF

sPut := CONCAT( CONCAT( CONCAT( sPrefix, sMessage ), sSource ), DWORD_TO_HEXSTR( nErrID AND 16#FFFF, 0, FALSE ) ); 

fbBuffer.A_AddTail( pBuffer:= ADR(buffer), cbBuffer:= SIZEOF(buffer),
					putValue:= sPut, bOk=>bOk, nCount=>nCount );
IF bOk THEN
	IF bLog THEN(* Log error message *)
		ADSLOGSTR( ADSLOG_MSGTYPE_ERROR OR ADSLOG_MSGTYPE_LOG, '%s', sPut );	
	END_IF
END_IF
END_ACTION

ACTION Message:
(* Adds new fifo entry *)
sPut := CONCAT( CONCAT( sPrefix, sMessage ), CONCAT( '::', HSOCKET_TO_STRING(hSocket) ) );
fbBuffer.A_AddTail( pBuffer:= ADR(buffer), cbBuffer:= SIZEOF(buffer),
					putValue:= sPut, bOk=>bOk, nCount=>nCount, cbSize=>ncbSize);
IF bOk THEN
	IF bLog THEN(* Log information message *)
		ADSLOGSTR( ADSLOG_MSGTYPE_HINT OR ADSLOG_MSGTYPE_LOG, '%s', sPut );	
	END_IF
END_IF
END_ACTION

ACTION Remove:
(* Removes oldest fifo entry *)
IF nCount = 0 THEN
	sGet := '';
	bOk := FALSE;
	RETURN;
END_IF

fbBuffer.A_RemoveHead( pBuffer:= ADR(buffer), cbBuffer:= SIZEOF(buffer),
						getValue=>sGet, bOk=>bOk, nCount=>nCount );
END_ACTION

END_FUNCTION_BLOCK

// ---- FunctionBlocks/Server/FB_ServerConnection.TcPOU
FUNCTION_BLOCK FB_ServerConnection
VAR_IN_OUT
	fbTx 			: FB_FrameFifo;(* TX fifo *)
	fbRx 			: FB_FrameFifo;(* RX fifo *)
	fbLog			: FB_LogFifo;(* Log message fifo *)
	hListener		: T_HSOCKET;(* Listener socket handle *)
	bReset			: BOOL;
END_VAR
VAR_INPUT
	sSrvNetID		: T_AmsNetID	:= '';(* TwinCAT TCP/IP server network address *)
	bEnable 		: BOOL 			:= FALSE;(* TRUE => connect and exchange data, FALSE => disconnect *)
	tReconnect 		: TIME 			:= T#1S;(* Accept new connection (reconnect) after this time *)
	bLog			: BOOL			:= FALSE;(* TRUE => Enable log message output, FALSE => Disable *)
	sPrefix			: STRING 		:= 'SERVERx::';(* Log message description string (allows the identification of log message source) *)
	bAllowConnect	: BOOL;
END_VAR
VAR_OUTPUT
	bConnecting		: BOOL;						(*Indicate that this server connection is attempting to connect*)
	bAccepted		: BOOL			:= FALSE;(* Accepted connection status *)
	TestBuffer 		: ARRAY[0..ServerControl.PLCPRJ_BUFFER_SIZE] OF BYTE;
END_VAR
VAR
	{attribute 'OPC.UA.DA' := '1'}
	fbAccept 		: FB_SocketAccept;
	fbClose			: FB_SocketClose;
	fbReceive		: FB_SocketReceive;
	fbSend			: FB_SocketSend;
	eStep			: E_ConnectionSteps;
	bSndBusy 		: BOOL;(* Tx state *)
	bRcvBusy 		: BOOL;(* Rx state *)
	bDisconnect		: BOOL;(* Disconnect flag, if set the socket will be closed *)

	fbAcceptTimer	: TON;(* Accept poll timer *)
	fbPollTimer		: TON;(* Receive poll timer *)
	fbRequestTimer	: TON;(* Request timeout timer *)
	
	rxBuffer		: ARRAY[0..ServerControl.PLCPRJ_BUFFER_SIZE] OF BYTE;
	sTxFrame		: T_MaxString;
	sRxFrame		: T_MaxString;
	cbReceived		: UDINT;
	nLenOfString	: UDINT;(* String length inclusive the null delimiter *)
	bEndOfString	: BOOL := FALSE;
END_VAR

(*
	Determine the current state of this connection
*)
CASE eStep OF
	(*
		IDLE connections test for Enable and Accepted to change states
		IDLE transitions to CONNECT_START when not accepted and to CLOSE_START when not enabled and accepted
		IDLE transitons to DATAEXCHANGE when enabled and accepted 
	*)
	eCONNECTION_STATE_IDLE:
		IF bEnable XOR bAccepted THEN
			IF bEnable THEN
				fbAcceptTimer( IN := TRUE );
				IF fbAcceptTimer.Q  AND bAllowConnect THEN
					
					fbTx.Clear( sPrefix := CONCAT( sPrefix, 'FB_FrameFifo(send)::' ), bLog := bLog );(* Clear send fifo *)
					fbRx.Clear( sPrefix := CONCAT( sPrefix, 'FB_FrameFifo(recv)::' ), bLog := bLog );(* Clear receiver fifo *)
					fbLog.Clear( sPrefix := sPrefix, bLog := bLog );(* Clear log fifo *)
					bSndBusy := FALSE;
					bRcvBusy := FALSE;
					bDisconnect := FALSE;
					cbReceived := 0;
					
					fbPollTimer( IN := FALSE, PT := T#0S );
					fbRequestTimer( IN := FALSE, PT := ServerControl.PLCPRJ_RECEIVE_TIMEOUT );
					fbAcceptTimer( IN := FALSE, PT := tReconnect );
					
					eStep := eCONNECTION_STATE_CONNECT_START;
				END_IF
			ELSE
				eStep := eCONNECTION_STATE_CLOSE_START;
			END_IF
		ELSIF bAccepted THEN
			eStep := eCONNECTION_STATE_DATAEXCHANGE;
		ELSE
			fbAcceptTimer( IN := FALSE, PT := T#0S );
		END_IF
	(*
		CONNECT_START transitions to CONNECT_WAIT after initiating an FB_SocketAccept call
		bConnecting is used to limit accept attempts to a single accept at a time
	*)
	eCONNECTION_STATE_CONNECT_START:
		fbAccept( bExecute := FALSE );
		fbAccept( sSrvNetID := sSrvNetID, 
					hListener := hListener, 
					bExecute:= TRUE );
		eStep := eCONNECTION_STATE_CONNECT_WAIT;
		bConnecting := TRUE;

	eCONNECTION_STATE_CONNECT_WAIT:
		fbAccept( bExecute := FALSE );
		IF NOT fbAccept.bBusy THEN
			bConnecting := FALSE;
			IF NOT fbAccept.bError THEN
				IF fbAccept.bAccepted THEN
					bAccepted := TRUE;
					fbLog.Message( sMessage := 'Connection accepted!', hSocket := fbAccept.hSocket );
				END_IF
				eStep := eCONNECTION_STATE_IDLE;
			ELSE
				fbLog.Error( sMessage := 'FB_SocketAccept()', nErrId := fbAccept.nErrId );
				eStep := eCONNECTION_STATE_ERROR;
			END_IF
		END_IF

	eCONNECTION_STATE_DATAEXCHANGE:(* Data exchange state *)
		bDisconnect := NOT bEnable OR bDisconnect;(* User/internal disconnect requested? *)
		IF bDisconnect AND NOT bSndBusy AND NOT bRcvBusy THEN
			bDisconnect := FALSE;
			eStep := eCONNECTION_STATE_CLOSE_START;(* Disconnect *)
		ELSE
	
			(* Send tx data *)
			IF NOT bDisconnect AND NOT bSndBusy THEN
				fbTx.RemoveHead( sGet => sTxFrame );(* Remove oldest string entry s*)
				IF fbTx.bOk THEN(* Success *)
					fbSend( bExecute := FALSE );
					fbSend(	sSrvNetID := sSrvNetID, 
							hSocket	:= fbAccept.hSocket,
							pSrc	:= ADR( sTxFrame ),
							cbLen	:= INT_TO_UDINT(LEN( sTxFrame )) (*+ 1*),(* String length inclusive the zero delimiter *)
							bExecute:= TRUE );
					bSndBusy := TRUE;

				END_IF
			ELSE
				fbSend( bExecute := FALSE );
				IF NOT fbSend.bBusy THEN
					bSndBusy := FALSE;
					IF fbSend.bError THEN
						fbLog.Error( sMessage := 'FB_SocketSend()', nErrId := fbSend.nErrId );
						bDisconnect := TRUE;(* Set flag *)
					END_IF
				END_IF
			END_IF
		
		
			(* Get rx data *)
			IF NOT bDisconnect AND NOT bRcvBusy THEN
				fbPollTimer( IN := TRUE );
				IF fbPollTimer.Q THEN
					fbPollTimer( IN := FALSE, PT := ServerControl.PLCPRJ_RECEIVE_POLLING_TIME );
					fbReceive( bExecute := FALSE );
					fbReceive( 	sSrvNetID := sSrvNetID, 
								hSocket	:= fbAccept.hSocket,
								pDest	:= ADR( rxBuffer ) + cbReceived,
								cbLen	:= SIZEOF( rxBuffer ) - cbReceived,
								bExecute:= TRUE );
					bRcvBusy := TRUE;
					
				END_IF
			ELSE
				fbReceive( bExecute := FALSE );
				IF NOT fbReceive.bBusy THEN
					bRcvBusy := FALSE;
					IF NOT fbReceive.bError THEN						
						IF (fbReceive.nRecBytes > 0) THEN(* Bytes received *)
						
							fbPollTimer( IN := FALSE, PT := T#0S ); (* Bytes received => increase the read (polling) speed *)
							fbRequestTimer( IN := FALSE );(* Bytes received => disable timeout check *)
							cbReceived 	:= cbReceived + fbReceive.nRecBytes;(* Calculate the number of received data bytes *)
		
							REPEAT
								
								(* Search for string end delimiter *)
								nLenOfString := 0;(* Reset string length *)
								bEndOfString := FALSE;
								REPEAT 
									IF rxBuffer[nLenOfString] = 3 THEN(* String end delimiter found *)
										bEndOfString := TRUE;

									END_IF
									nLenOfString := nLenOfString + 1;
								UNTIL bEndOfString OR (nLenOfString >= cbReceived)
								END_REPEAT
								
								IF bEndOfString THEN
									MEMSET( ADR( sRxFrame ), 0, SIZEOF( sRxFrame ) );
									MEMCPY(  ADR( sRxFrame ), ADR( rxBuffer ), MIN( SIZEOF(sRxFrame), nLenOfString ) );(* Copy the received string to the output variable (inclusive the end delimiter) *)
									MEMMOVE( ADR( rxBuffer ), ADR( rxBuffer[nLenOfString] ), cbReceived - nLenOfString  );(* Move the reamaining data bytes *)
									cbReceived := cbReceived - nLenOfString;(* Recalculate the reamaining data byte length *)
								
									fbRx.AddTail( sPut := sRxFrame );(* Put received message to the rx fifo *)
									IF NOT fbRx.bOk THEN
										fbLog.Error( sMessage := 'FB_FrameFifo(receiver)', nErrID := ServerControl.PLCPRJ_ERROR_RECFIFO_OVERFLOW );
										bDisconnect := TRUE;(* Set flag *)
										RETURN;
									END_IF
								END_IF

							UNTIL NOT bEndOfString OR (cbReceived = 0)
							END_REPEAT
		
						ELSE(* No bytes received *)
							fbRequestTimer( IN := TRUE, PT := ServerControl.PLCPRJ_RECEIVE_TIMEOUT );(* No bytes received => enable timeout check *)
							IF fbRequestTimer.Q THEN (* Timeout error*)
								fbRequestTimer( IN := FALSE );
								fbLog.Error( sMessage := 'FB_SocketReceive()', nErrID := ServerControl.PLCPRJ_ERROR_RECEIVE_TIMEOUT );
								bDisconnect := TRUE;(* Set flag *)
							END_IF
						END_IF
						
					ELSE(* Receive error *)
						fbLog.Error( sMessage := 'FB_SocketReceive()', nErrId := fbReceive.nErrId );
						bDisconnect := TRUE;(* Set flag *)
					END_IF
				END_IF(* IF NOT fbReceive.bBusy THEN *)
				
			END_IF(* IF NOT bDisconnect AND NOT bRcvBusy THEN *)
		
		END_IF(* IF bDisconnect AND NOT bSndBusy AND NOT bRcvBusy THEN *)
	
	

	eCONNECTION_STATE_CLOSE_START:
		fbLog.Message( sMessage := 'Closing connection!', hSocket := fbAccept.hSocket );
		fbClose( bExecute := FALSE );
		fbClose( sSrvNetID := sSrvNetID, hSocket:= fbAccept.hSocket, bExecute:= TRUE );
		eStep := eCONNECTION_STATE_CLOSE_WAIT;

	eCONNECTION_STATE_CLOSE_WAIT:
		fbClose( bExecute := FALSE );
		IF NOT fbClose.bBusy THEN
			bAccepted := FALSE;
			IF NOT fbClose.bError THEN
				eStep := eCONNECTION_STATE_IDLE;
			ELSE
				fbLog.Error( sMessage := 'FB_SocketClose(accepted)', nErrId := fbClose.nErrId );
				eStep := eCONNECTION_STATE_ERROR;
			END_IF
		END_IF

	eCONNECTION_STATE_ERROR:
		IF bAccepted THEN
			eStep := eCONNECTION_STATE_CLOSE_START;
		ELSE
			eStep := eCONNECTION_STATE_IDLE;
		END_IF

END_CASE

END_FUNCTION_BLOCK

// ---- FunctionBlocks/Utils/IncIndex.TcPOU
FUNCTION IncIndex : INT
VAR_INPUT
	IDX:	INT;		// Index to be incremented
	IdxMIN:	INT;		// Min Value for index	
	IdxMAX:	INT;		// Max Value for index
END_VAR
VAR
END_VAR

IF IDX < IdxMAX THEN
	IncIndex := IDX + 1; 
ELSIF IDX = IdxMAX THEN
	IncIndex := IdxMIN;
ELSIF IDX < IdxMIN OR IDX > IdxMAX THEN
	 IncIndex := IdxMIN;
END_IF

END_FUNCTION

// ---- POUs/Log_Diverts_P2140.TcPOU
PROGRAM Log_Diverts_P2140
VAR
	r_DivertExtend			: ARRAY [1..16] OF R_TRIG;
	f_DivertExtend			: ARRAY [1..16] OF F_TRIG;
	r_ConfirmPE				: ARRAY [1..16] OF R_TRIG;
	f_ConfirmPE				: ARRAY [1..16] OF F_TRIG;
	sMessage				: STRING;
END_VAR

// Divert 1
r_DivertExtend[1](CLK := Sorter.aSorterDiverts_P2140[1].Output1);
f_DivertExtend[1](CLK := Sorter.aSorterDiverts_P2140[1].Output1);

IF r_DivertExtend[1].Q THEN
	IF .nDivertLogEnable.DIVERT1 THEN
		ADSLOGSTR( msgCtrlMask := ADSLOG_MSGTYPE_HINT OR ADSLOG_MSGTYPE_LOG
			, msgFmtStr := 'Extend Divert 1 : %s'
			, strArg := UDINT_TO_STRING(Sorter.st_SorterEncoder_P2140.CurrentCount)); 
	END_IF;
END_IF
IF f_DivertExtend[1].Q THEN
	IF .nDivertLogEnable.DIVERT1 THEN
		ADSLOGSTR( msgCtrlMask := ADSLOG_MSGTYPE_HINT OR ADSLOG_MSGTYPE_LOG
			, msgFmtStr := 'Retract Divert 1 : %s'
			, strArg := UDINT_TO_STRING(Sorter.st_SorterEncoder_P2140.CurrentCount)); 
	END_IF;
END_IF

// Confirm 1
r_ConfirmPE[1](CLK := Sorter.aSorterDiverts_P2140[1].ConfirmPE);
f_ConfirmPE[1](CLK := Sorter.aSorterDiverts_P2140[1].ConfirmPE);

IF r_ConfirmPE[1].Q THEN
	IF .nDivertLogEnable.CONFIRM1 THEN
		ADSLOGSTR( msgCtrlMask := ADSLOG_MSGTYPE_HINT OR ADSLOG_MSGTYPE_LOG
			, msgFmtStr := 'Confirm PE 1 Blocked: %s'
			, strArg := UDINT_TO_STRING(Sorter.st_SorterEncoder_P2140.CurrentCount)); 
	END_IF;
END_IF
IF f_ConfirmPE[1].Q THEN
	IF .nDivertLogEnable.CONFIRM1 THEN
		ADSLOGSTR( msgCtrlMask := ADSLOG_MSGTYPE_HINT OR ADSLOG_MSGTYPE_LOG
			, msgFmtStr := 'Confirm PE 1 Clear: %s'
			, strArg := UDINT_TO_STRING(Sorter.st_SorterEncoder_P2140.CurrentCount)); 
	END_IF;
END_IF

// Divert 2
r_DivertExtend[2](CLK := Sorter.aSorterDiverts_P2140[2].Output1);
f_DivertExtend[2](CLK := Sorter.aSorterDiverts_P2140[2].Output1);

IF r_DivertExtend[2].Q THEN
	IF .nDivertLogEnable.DIVERT2 THEN
		ADSLOGSTR( msgCtrlMask := ADSLOG_MSGTYPE_HINT OR ADSLOG_MSGTYPE_LOG
			, msgFmtStr := 'Extend Divert 2: %s'
			, strArg := UDINT_TO_STRING(Sorter.st_SorterEncoder_P2140.CurrentCount)); 
	END_IF;
END_IF
IF f_DivertExtend[2].Q THEN
	IF .nDivertLogEnable.DIVERT2 THEN
		ADSLOGSTR( msgCtrlMask := ADSLOG_MSGTYPE_HINT OR ADSLOG_MSGTYPE_LOG
			, msgFmtStr := 'Retract Divert 2: %s'
			, strArg := UDINT_TO_STRING(Sorter.st_SorterEncoder_P2140.CurrentCount)); 
	END_IF;
END_IF

// Confirm 2
r_ConfirmPE[2](CLK := Sorter.aSorterDiverts_P2140[2].ConfirmPE);
f_ConfirmPE[2](CLK := Sorter.aSorterDiverts_P2140[2].ConfirmPE);

IF r_ConfirmPE[2].Q THEN
	IF .nDivertLogEnable.CONFIRM2 THEN
		ADSLOGSTR( msgCtrlMask := ADSLOG_MSGTYPE_HINT OR ADSLOG_MSGTYPE_LOG
			, msgFmtStr := 'Confirm PE 2 Blocked: %s'
			, strArg := UDINT_TO_STRING(Sorter.st_SorterEncoder_P2140.CurrentCount)); 
	END_IF;
END_IF
IF f_ConfirmPE[2].Q THEN
	IF .nDivertLogEnable.CONFIRM2 THEN
		ADSLOGSTR( msgCtrlMask := ADSLOG_MSGTYPE_HINT OR ADSLOG_MSGTYPE_LOG
			, msgFmtStr := 'Confirm PE 2 Clear: %s'
			, strArg := UDINT_TO_STRING(Sorter.st_SorterEncoder_P2140.CurrentCount)); 
	END_IF
END_IF

END_PROGRAM

// ---- POUs/Log_Diverts_P2150.TcPOU
PROGRAM Log_Diverts_P2150
VAR
	r_DivertExtend			: ARRAY [1..16] OF R_TRIG;
	f_DivertExtend			: ARRAY [1..16] OF F_TRIG;
	r_ConfirmPE				: ARRAY [1..16] OF R_TRIG;
	f_ConfirmPE				: ARRAY [1..16] OF F_TRIG;
	sMessage				: STRING;
END_VAR

// Divert 1
r_DivertExtend[1](CLK := Sorter.aSorterDiverts_P2150[1].Output1);
f_DivertExtend[1](CLK := Sorter.aSorterDiverts_P2150[1].Output1);

IF r_DivertExtend[1].Q THEN
	IF .nDivertLogEnable.DIVERT1 THEN
		ADSLOGSTR( msgCtrlMask := ADSLOG_MSGTYPE_HINT OR ADSLOG_MSGTYPE_LOG
			, msgFmtStr := 'Extend Divert 1 : %s'
			, strArg := UDINT_TO_STRING(Sorter.st_SorterEncoder_P2150.CurrentCount)); 
	END_IF;
END_IF
IF f_DivertExtend[1].Q THEN
	IF .nDivertLogEnable.DIVERT1 THEN
		ADSLOGSTR( msgCtrlMask := ADSLOG_MSGTYPE_HINT OR ADSLOG_MSGTYPE_LOG
			, msgFmtStr := 'Retract Divert 1 : %s'
			, strArg := UDINT_TO_STRING(Sorter.st_SorterEncoder_P2150.CurrentCount)); 
	END_IF;
END_IF

// Confirm 1
r_ConfirmPE[1](CLK := Sorter.aSorterDiverts_P2150[1].ConfirmPE);
f_ConfirmPE[1](CLK := Sorter.aSorterDiverts_P2150[1].ConfirmPE);

IF r_ConfirmPE[1].Q THEN
	IF .nDivertLogEnable.CONFIRM1 THEN
		ADSLOGSTR( msgCtrlMask := ADSLOG_MSGTYPE_HINT OR ADSLOG_MSGTYPE_LOG
			, msgFmtStr := 'Confirm PE 1 Blocked: %s'
			, strArg := UDINT_TO_STRING(Sorter.st_SorterEncoder_P2150.CurrentCount)); 
	END_IF;
END_IF
IF f_ConfirmPE[1].Q THEN
	IF .nDivertLogEnable.CONFIRM1 THEN
		ADSLOGSTR( msgCtrlMask := ADSLOG_MSGTYPE_HINT OR ADSLOG_MSGTYPE_LOG
			, msgFmtStr := 'Confirm PE 1 Clear: %s'
			, strArg := UDINT_TO_STRING(Sorter.st_SorterEncoder_P2150.CurrentCount)); 
	END_IF;
END_IF

// Divert 2
r_DivertExtend[2](CLK := Sorter.aSorterDiverts_P2150[2].Output1);
f_DivertExtend[2](CLK := Sorter.aSorterDiverts_P2150[2].Output1);

IF r_DivertExtend[2].Q THEN
	IF .nDivertLogEnable.DIVERT2 THEN
		ADSLOGSTR( msgCtrlMask := ADSLOG_MSGTYPE_HINT OR ADSLOG_MSGTYPE_LOG
			, msgFmtStr := 'Extend Divert 2: %s'
			, strArg := UDINT_TO_STRING(Sorter.st_SorterEncoder_P2150.CurrentCount)); 
	END_IF;
END_IF
IF f_DivertExtend[2].Q THEN
	IF .nDivertLogEnable.DIVERT2 THEN
		ADSLOGSTR( msgCtrlMask := ADSLOG_MSGTYPE_HINT OR ADSLOG_MSGTYPE_LOG
			, msgFmtStr := 'Retract Divert 2: %s'
			, strArg := UDINT_TO_STRING(Sorter.st_SorterEncoder_P2150.CurrentCount)); 
	END_IF;
END_IF

// Confirm 2
r_ConfirmPE[2](CLK := Sorter.aSorterDiverts_P2150[2].ConfirmPE);
f_ConfirmPE[2](CLK := Sorter.aSorterDiverts_P2150[2].ConfirmPE);

IF r_ConfirmPE[2].Q THEN
	IF .nDivertLogEnable.CONFIRM2 THEN
		ADSLOGSTR( msgCtrlMask := ADSLOG_MSGTYPE_HINT OR ADSLOG_MSGTYPE_LOG
			, msgFmtStr := 'Confirm PE 2 Blocked: %s'
			, strArg := UDINT_TO_STRING(Sorter.st_SorterEncoder_P2150.CurrentCount)); 
	END_IF;
END_IF
IF f_ConfirmPE[2].Q THEN
	IF .nDivertLogEnable.CONFIRM2 THEN
		ADSLOGSTR( msgCtrlMask := ADSLOG_MSGTYPE_HINT OR ADSLOG_MSGTYPE_LOG
			, msgFmtStr := 'Confirm PE 2 Clear: %s'
			, strArg := UDINT_TO_STRING(Sorter.st_SorterEncoder_P2150.CurrentCount)); 
	END_IF
END_IF

// Sorter Discharge "Divert"
// Divert 3
r_DivertExtend[3](CLK := Sorter.aSorterDiverts_P2150[3].Output1);
f_DivertExtend[3](CLK := Sorter.aSorterDiverts_P2150[3].Output1);

IF r_DivertExtend[3].Q THEN
	IF .nDivertLogEnable.DIVERT3 THEN
		ADSLOGSTR( msgCtrlMask := ADSLOG_MSGTYPE_HINT OR ADSLOG_MSGTYPE_LOG
			, msgFmtStr := 'Extend Divert 3: %s'
			, strArg := UDINT_TO_STRING(Sorter.st_SorterEncoder_P2150.CurrentCount)); 
	END_IF;
END_IF
IF f_DivertExtend[3].Q THEN
	IF .nDivertLogEnable.DIVERT3 THEN
		ADSLOGSTR( msgCtrlMask := ADSLOG_MSGTYPE_HINT OR ADSLOG_MSGTYPE_LOG
			, msgFmtStr := 'Retract Divert 3: %s'
			, strArg := UDINT_TO_STRING(Sorter.st_SorterEncoder_P2150.CurrentCount)); 
	END_IF;
END_IF

// Confirm 3
r_ConfirmPE[3](CLK := Sorter.aSorterDiverts_P2150[3].ConfirmPE);
f_ConfirmPE[3](CLK := Sorter.aSorterDiverts_P2150[3].ConfirmPE);

IF r_ConfirmPE[3].Q THEN
	IF .nDivertLogEnable.CONFIRM3 THEN
		ADSLOGSTR( msgCtrlMask := ADSLOG_MSGTYPE_HINT OR ADSLOG_MSGTYPE_LOG
			, msgFmtStr := 'Confirm PE 3 Blocked: %s'
			, strArg := UDINT_TO_STRING(Sorter.st_SorterEncoder_P2150.CurrentCount)); 
	END_IF;
END_IF
IF f_ConfirmPE[3].Q THEN
	IF .nDivertLogEnable.CONFIRM3 THEN
		ADSLOGSTR( msgCtrlMask := ADSLOG_MSGTYPE_HINT OR ADSLOG_MSGTYPE_LOG
			, msgFmtStr := 'Confirm PE 3 Clear: %s'
			, strArg := UDINT_TO_STRING(Sorter.st_SorterEncoder_P2150.CurrentCount)); 
	END_IF
END_IF

// Sorter Discharge "Divert"
// Divert 4
r_DivertExtend[4](CLK := Sorter.aSorterDiverts_P2150[4].Output1);
f_DivertExtend[4](CLK := Sorter.aSorterDiverts_P2150[4].Output1);

IF r_DivertExtend[4].Q THEN
	IF .nDivertLogEnable.DIVERT4 THEN
		ADSLOGSTR( msgCtrlMask := ADSLOG_MSGTYPE_HINT OR ADSLOG_MSGTYPE_LOG
			, msgFmtStr := 'Extend Divert 4: %s'
			, strArg := UDINT_TO_STRING(Sorter.st_SorterEncoder_P2150.CurrentCount)); 
	END_IF;
END_IF
IF f_DivertExtend[4].Q THEN
	IF .nDivertLogEnable.DIVERT4 THEN
		ADSLOGSTR( msgCtrlMask := ADSLOG_MSGTYPE_HINT OR ADSLOG_MSGTYPE_LOG
			, msgFmtStr := 'Retract Divert 4: %s'
			, strArg := UDINT_TO_STRING(Sorter.st_SorterEncoder_P2150.CurrentCount)); 
	END_IF;
END_IF

// Confirm 4
r_ConfirmPE[4](CLK := Sorter.aSorterDiverts_P2150[4].ConfirmPE);
f_ConfirmPE[4](CLK := Sorter.aSorterDiverts_P2150[4].ConfirmPE);

IF r_ConfirmPE[4].Q THEN
	IF .nDivertLogEnable.CONFIRM4 THEN
		ADSLOGSTR( msgCtrlMask := ADSLOG_MSGTYPE_HINT OR ADSLOG_MSGTYPE_LOG
			, msgFmtStr := 'Confirm PE 4 Blocked: %s'
			, strArg := UDINT_TO_STRING(Sorter.st_SorterEncoder_P2150.CurrentCount)); 
	END_IF;
END_IF
IF f_ConfirmPE[4].Q THEN
	IF .nDivertLogEnable.CONFIRM4 THEN
		ADSLOGSTR( msgCtrlMask := ADSLOG_MSGTYPE_HINT OR ADSLOG_MSGTYPE_LOG
			, msgFmtStr := 'Confirm PE 4 Clear: %s'
			, strArg := UDINT_TO_STRING(Sorter.st_SorterEncoder_P2150.CurrentCount)); 
	END_IF
END_IF	

// Sorter Discharge "Divert"
// Divert 5
r_DivertExtend[5](CLK := Sorter.aSorterDiverts_P2150[5].Output1);
f_DivertExtend[5](CLK := Sorter.aSorterDiverts_P2150[5].Output1);

IF r_DivertExtend[5].Q THEN
	IF .nDivertLogEnable.DIVERT5 THEN
		ADSLOGSTR( msgCtrlMask := ADSLOG_MSGTYPE_HINT OR ADSLOG_MSGTYPE_LOG
			, msgFmtStr := 'Extend Divert 5: %s'
			, strArg := UDINT_TO_STRING(Sorter.st_SorterEncoder_P2150.CurrentCount)); 
	END_IF;
END_IF
IF f_DivertExtend[5].Q THEN
	IF .nDivertLogEnable.DIVERT5 THEN
		ADSLOGSTR( msgCtrlMask := ADSLOG_MSGTYPE_HINT OR ADSLOG_MSGTYPE_LOG
			, msgFmtStr := 'Retract Divert 5: %s'
			, strArg := UDINT_TO_STRING(Sorter.st_SorterEncoder_P2150.CurrentCount)); 
	END_IF;
END_IF

// Confirm 5
r_ConfirmPE[5](CLK := Sorter.aSorterDiverts_P2150[5].ConfirmPE);
f_ConfirmPE[5](CLK := Sorter.aSorterDiverts_P2150[5].ConfirmPE);

IF r_ConfirmPE[5].Q THEN
	IF .nDivertLogEnable.CONFIRM5 THEN
		ADSLOGSTR( msgCtrlMask := ADSLOG_MSGTYPE_HINT OR ADSLOG_MSGTYPE_LOG
			, msgFmtStr := 'Confirm PE 5 Blocked: %s'
			, strArg := UDINT_TO_STRING(Sorter.st_SorterEncoder_P2150.CurrentCount)); 
	END_IF;
END_IF
IF f_ConfirmPE[5].Q THEN
	IF .nDivertLogEnable.CONFIRM5 THEN
		ADSLOGSTR( msgCtrlMask := ADSLOG_MSGTYPE_HINT OR ADSLOG_MSGTYPE_LOG
			, msgFmtStr := 'Confirm PE 5 Clear: %s'
			, strArg := UDINT_TO_STRING(Sorter.st_SorterEncoder_P2150.CurrentCount)); 
	END_IF
END_IF

END_PROGRAM

// ---- POUs/P_PulseCountDist.TcPOU
PROGRAM P_PulseCountDist
VAR
	EncoderValue : UDINT;
	StartValue: UDINT;
	EndValue: UDINT;
	Reading: BOOL;
	TotalCounts: UDINT;
	ReadCount: UDINT;
	ReadSum: UDINT;
	ReadAvg: REAL;
	Reset: BOOL;
	Timer: TON;
	TimeElapsed: REAL;
	Distance : REAL;
	Speed_ips : REAL;
	Speed_fps : REAL;
	Speed_fpm : REAL;
	DistperCount :	REAL;
	TestStart: R_TRIG;
	TestEnd: R_TRIG;
END_VAR

VAR CONSTANT
	EncoderMax: UDINT := Sorter.SORTERENCODERMAX_P2150;
END_VAR

// Uncomment to get pulse counts for a distance
TestStart(CLK:= (* Start photo eye goes here --> *) Photoeyes.PE_11291.Out);
TestEnd(CLK:= (* End photo eye goes here --> *) Photoeyes.PE_10302.Out);
EncoderValue := GVL_IO.ENC_9031_Raw;

Timer(IN:= Reading, PT:= T#1H, Q=> , ET=> );

IF Reset THEN
	ReadCount := 0;	
	ReadSum := 0;
	ReadAvg := 0;
	Reset := FALSE;
END_IF

IF TestStart.Q THEN 
	StartValue := EncoderValue;
	Reading := TRUE;
	ReadCount := ReadCount +1;
END_IF

IF Reading THEN
	TimeElapsed := (TIME_TO_REAL(Timer.ET))/1000;
END_IF

IF TestEnd.Q THEN 
	EndValue := EncoderValue;
	IF EndValue < StartValue THEN
		TotalCounts := EncoderMax - StartValue;
		TotalCounts := TotalCounts + EndValue;
	ELSE
  		TotalCounts := (EndValue-StartValue);
	END_IF
	
	ReadSum := ReadSum + TotalCounts;
	IF  ReadCount > 0 THEN 
		ReadAvg := UDINT_TO_REAL(ReadSum)/UDINT_TO_REAL(ReadCount);
	END_IF
	 
